ACTION SubModules_Action:
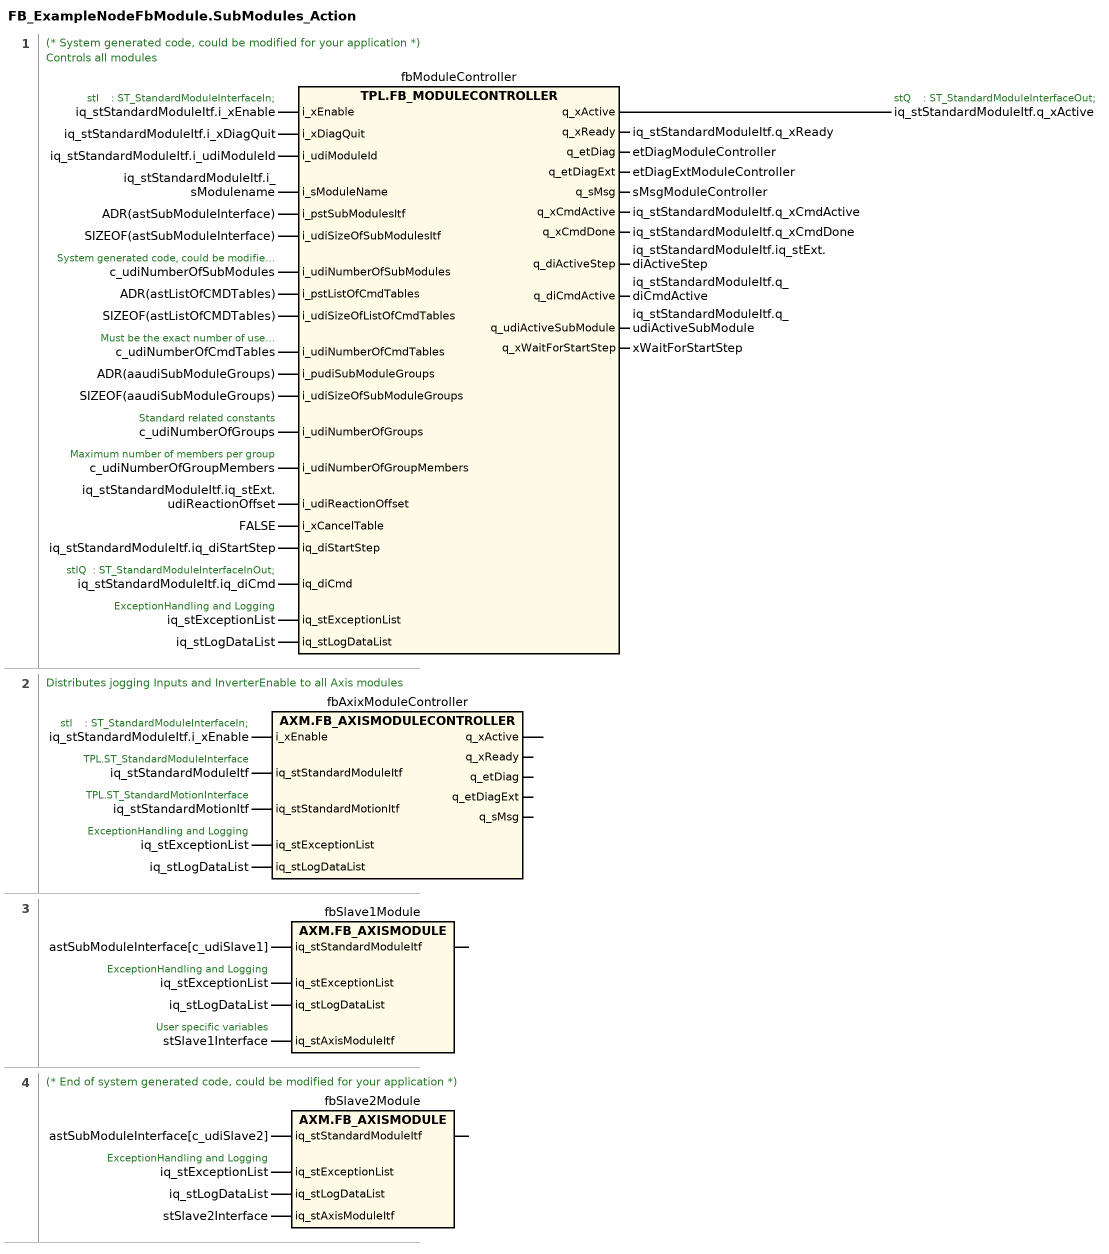
// NETWORK 1
// 					(* System generated code, could be modified for your application *)
// Controls all modules
//
//   fbModuleController: Modules related variables
//   iq_stStandardModuleItf.i_xEnable: stI : ST_StandardModuleInterfaceIn;
//   c_udiNumberOfSubModules: System generated code, could be modified for your application
//   c_udiNumberOfCmdTables: Must be the exact number of used CMDTables!
//   c_udiNumberOfGroups: Standard related constants
//   c_udiNumberOfGroupMembers: Maximum number of members per group
//   iq_stStandardModuleItf.iq_diCmd: stIQ : ST_StandardModuleInterfaceInOut;
//   iq_stExceptionList: ExceptionHandling and Logging
//   iq_stStandardModuleItf.q_xActive: stQ : ST_StandardModuleInterfaceOut;
fbModuleController(
    i_xEnable := iq_stStandardModuleItf.i_xEnable,
    i_xDiagQuit := iq_stStandardModuleItf.i_xDiagQuit,
    i_udiModuleId := iq_stStandardModuleItf.i_udiModuleId,
    i_sModuleName := iq_stStandardModuleItf.i_sModulename,
    i_pstSubModulesItf := ADR(astSubModuleInterface),
    i_udiSizeOfSubModulesItf := SIZEOF(astSubModuleInterface),
    i_udiNumberOfSubModules := c_udiNumberOfSubModules,
    i_pstListOfCmdTables := ADR(astListOfCMDTables),
    i_udiSizeOfListOfCmdTables := SIZEOF(astListOfCMDTables),
    i_udiNumberOfCmdTables := c_udiNumberOfCmdTables,
    i_pudiSubModuleGroups := ADR(aaudiSubModuleGroups),
    i_udiSizeOfSubModuleGroups := SIZEOF(aaudiSubModuleGroups),
    i_udiNumberOfGroups := c_udiNumberOfGroups,
    i_udiNumberOfGroupMembers := c_udiNumberOfGroupMembers,
    i_udiReactionOffset := iq_stStandardModuleItf.iq_stExt.udiReactionOffset,
    i_xCancelTable := FALSE,
    iq_diStartStep := iq_stStandardModuleItf.iq_diStartStep,
    iq_diCmd := iq_stStandardModuleItf.iq_diCmd,
    iq_stExceptionList := iq_stExceptionList,
    iq_stLogDataList := iq_stLogDataList,
    q_xReady => iq_stStandardModuleItf.q_xReady,
    q_etDiag => etDiagModuleController,
    q_etDiagExt => etDiagExtModuleController,
    q_sMsg => sMsgModuleController,
    q_xCmdActive => iq_stStandardModuleItf.q_xCmdActive,
    q_xCmdDone => iq_stStandardModuleItf.q_xCmdDone,
    q_diActiveStep => iq_stStandardModuleItf.iq_stExt.diActiveStep,
    q_diCmdActive => iq_stStandardModuleItf.q_diCmdActive,
    q_udiActiveSubModule => iq_stStandardModuleItf.q_udiActiveSubModule,
    q_xWaitForStartStep => xWaitForStartStep); // TPL.FB_MODULECONTROLLER
iq_stStandardModuleItf.q_xActive := fbModuleController.q_xActive;

// NETWORK 2
// Distributes jogging Inputs and InverterEnable to all Axis modules
//   iq_stStandardModuleItf.i_xEnable: stI : ST_StandardModuleInterfaceIn;
//   iq_stStandardModuleItf: TPL.ST_StandardModuleInterface
//   iq_stStandardMotionItf: TPL.ST_StandardMotionInterface
//   iq_stExceptionList: ExceptionHandling and Logging
fbAxixModuleController(
    i_xEnable := iq_stStandardModuleItf.i_xEnable,
    iq_stStandardModuleItf := iq_stStandardModuleItf,
    iq_stStandardMotionItf := iq_stStandardMotionItf,
    iq_stExceptionList := iq_stExceptionList,
    iq_stLogDataList := iq_stLogDataList); // AXM.FB_AXISMODULECONTROLLER

// NETWORK 3
//   iq_stExceptionList: ExceptionHandling and Logging
//   stSlave1Interface: User specific variables
fbSlave1Module(
    iq_stStandardModuleItf := astSubModuleInterface[c_udiSlave1],
    iq_stExceptionList := iq_stExceptionList,
    iq_stLogDataList := iq_stLogDataList,
    iq_stAxisModuleItf := stSlave1Interface); // AXM.FB_AXISMODULE

// NETWORK 4
// (* End of system generated code, could be modified for your application *)
//   iq_stExceptionList: ExceptionHandling and Logging
fbSlave2Module(
    iq_stStandardModuleItf := astSubModuleInterface[c_udiSlave2],
    iq_stExceptionList := iq_stExceptionList,
    iq_stLogDataList := iq_stLogDataList,
    iq_stAxisModuleItf := stSlave2Interface); // AXM.FB_AXISMODULE
END_ACTION

ACTION UpdateStructs:
(* System generated code, do not change without consulting 'Schneider Electric Automation GmbH' - otherwise you risk instability!!!*)
fbDetectOnlineChange(	i_xEnable	:= TRUE, 
						i_xDetect	:= TRUE, 
						q_xActive	=> xDetectOnlineChangeActive, 
						q_xReady	=> xDetectOnlineChangeReady, 
						q_etDiag	=> etDetectOnlineChangeDiag, 
						q_etDiagExt	=> etDetectOnlineChangeDiagExt, 
						q_sMsg		=> sDetectOnlineChangeMsg, 
						q_xChange	=> );
						
IF(NOT fbDetectOnlineChange.q_xChange) THEN
	RETURN;
END_IF

iq_stStandardModuleItf.iq_stExt.udiNumberOfSubModules 	:= c_udiNumberOfSubModules;
iq_stStandardModuleItf.iq_stExt.dwSubModulesItf		 	:= ADR(astSubModuleInterface);
iq_stStandardModuleItf.iq_stExt.pdwSubModulesAddItf 	:= ADR(adwSubModuleAddInterfaces);
iq_stStandardModuleItf.iq_stExt.pstListOfCmdTables		:= ADR(astListOfCmdTables);
iq_stStandardModuleItf.iq_stExt.udiNumberOfCmdTables	:= c_udiNumberOfCmdTables;
(* End of system generated code, do not change without consulting 'Schneider Electric Automation GmbH' - otherwise you risk instability!!!*)

(* System generated code, could be modified for your application *)
xUpdateStructsException := FALSE;

(*****************************************************************************************************************************************************)
(* Update CmdTable - Prepare *)

TPL.FC_UpdateCmdTableListElement(	i_pstListofCmdTables	:= ADR(astListOfCmdTables),
									i_udiNumberOfCmdTables	:= c_udiNumberOfCmdTables,
									i_diCmd					:= ET_Cmd.Prepare,
									i_pstCmdTable			:= ADR(astPrepareTable),
									q_etDiag				=> etDiag,
									q_etDiagExt				=> etDiagExtTPL);
									
IF etDiag <> GD.ET_Diag.Ok AND NOT xUpdateStructsException THEN
	xUpdateStructsException := TRUE;
	
	stUpdateStructsException.sMsg := PDL.FC_MultiConcat(i_sString1 := 'Update CmdTable: Prepare - ', 
														i_sString2 := GD.FC_EtDiagToString(i_etDiag := etDiag), 
														i_sString3 := ' - ', 
														i_sString4 := TPL.FC_EtDiagExtToString(i_etDiagExt := etDiagExtTPL));
END_IF										

(*****************************************************************************************************************************************************)
(* Update CmdTable - Auto *)

TPL.FC_UpdateCmdTableListElement(	i_pstListofCmdTables	:= ADR(astListOfCmdTables),
									i_udiNumberOfCmdTables	:= c_udiNumberOfCmdTables,
									i_diCmd					:= ET_Cmd.Auto,
									i_pstCmdTable			:= ADR(astAutoTable),
									q_etDiag				=> etDiag,
									q_etDiagExt				=> etDiagExtTPL);
									
IF etDiag <> GD.ET_Diag.Ok AND NOT xUpdateStructsException THEN
	xUpdateStructsException := TRUE;
	
	stUpdateStructsException.sMsg := PDL.FC_MultiConcat(i_sString1 := 'Update CmdTable: Auto - ', 
														i_sString2 := GD.FC_EtDiagToString(i_etDiag := etDiag), 
														i_sString3 := ' - ', 
														i_sString4 := TPL.FC_EtDiagExtToString(i_etDiagExt := etDiagExtTPL));
END_IF		

(*****************************************************************************************************************************************************)
(* Update CmdTable - Manual *)

TPL.FC_UpdateCmdTableListElement(	i_pstListofCmdTables	:= ADR(astListOfCmdTables),
									i_udiNumberOfCmdTables	:= c_udiNumberOfCmdTables,
									i_diCmd					:= ET_Cmd.Manual,
									i_pstCmdTable			:= ADR(astManualTable),
									q_etDiag				=> etDiag,
									q_etDiagExt				=> etDiagExtTPL);
									
IF etDiag <> GD.ET_Diag.Ok AND NOT xUpdateStructsException THEN
	xUpdateStructsException := TRUE;
	
	stUpdateStructsException.sMsg := PDL.FC_MultiConcat(i_sString1 := 'Update CmdTable: Manual - ', 
														i_sString2 := GD.FC_EtDiagToString(i_etDiag := etDiag), 
														i_sString3 := ' - ', 
														i_sString4 := TPL.FC_EtDiagExtToString(i_etDiagExt := etDiagExtTPL));
END_IF		

(*****************************************************************************************************************************************************)
(* Update CmdTable - Stop *)

TPL.FC_UpdateCmdTableListElement(	i_pstListofCmdTables	:= ADR(astListOfCmdTables),
									i_udiNumberOfCmdTables	:= c_udiNumberOfCmdTables,
									i_diCmd					:= ET_Cmd.Stop,
									i_pstCmdTable			:= ADR(astStopTable),
									q_etDiag				=> etDiag,
									q_etDiagExt				=> etDiagExtTPL);
									
IF etDiag <> GD.ET_Diag.Ok AND NOT xUpdateStructsException THEN
	xUpdateStructsException := TRUE;
	
	stUpdateStructsException.sMsg := PDL.FC_MultiConcat(i_sString1 := 'Update CmdTable: Stop - ', 
														i_sString2 := GD.FC_EtDiagToString(i_etDiag := etDiag), 
														i_sString3 := ' - ', 
														i_sString4 := TPL.FC_EtDiagExtToString(i_etDiagExt := etDiagExtTPL));
END_IF		

(*****************************************************************************************************************************************************)
(* Update CmdTable - Start *)

TPL.FC_UpdateCmdTableListElement(	i_pstListofCmdTables	:= ADR(astListOfCmdTables),
									i_udiNumberOfCmdTables	:= c_udiNumberOfCmdTables,
									i_diCmd					:= ET_Cmd.Start,
									i_pstCmdTable			:= ADR(astStartTable),
									q_etDiag				=> etDiag,
									q_etDiagExt				=> etDiagExtTPL);
									
IF etDiag <> GD.ET_Diag.Ok AND NOT xUpdateStructsException THEN
	xUpdateStructsException := TRUE;
	
	stUpdateStructsException.sMsg := PDL.FC_MultiConcat(i_sString1 := 'Update CmdTable: Start - ', 
														i_sString2 := GD.FC_EtDiagToString(i_etDiag := etDiag), 
														i_sString3 := ' - ', 
														i_sString4 := TPL.FC_EtDiagExtToString(i_etDiagExt := etDiagExtTPL));
END_IF		

(*****************************************************************************************************************************************************)
(* Update CmdTable - Abort *)

TPL.FC_UpdateCmdTableListElement(	i_pstListofCmdTables	:= ADR(astListOfCmdTables),
									i_udiNumberOfCmdTables	:= c_udiNumberOfCmdTables,
									i_diCmd					:= ET_Cmd.Abort,
									i_pstCmdTable			:= ADR(astAbortTable),
									q_etDiag				=> etDiag,
									q_etDiagExt				=> etDiagExtTPL);
									
IF etDiag <> GD.ET_Diag.Ok AND NOT xUpdateStructsException THEN
	xUpdateStructsException := TRUE;
	
	stUpdateStructsException.sMsg := PDL.FC_MultiConcat(i_sString1 := 'Update CmdTable: Abort - ', 
														i_sString2 := GD.FC_EtDiagToString(i_etDiag := etDiag), 
														i_sString3 := ' - ', 
														i_sString4 := TPL.FC_EtDiagExtToString(i_etDiagExt := etDiagExtTPL));
END_IF		

(*****************************************************************************************************************************************************)
(* Update CmdTable - Hold *)

TPL.FC_UpdateCmdTableListElement(	i_pstListofCmdTables	:= ADR(astListOfCmdTables),
									i_udiNumberOfCmdTables	:= c_udiNumberOfCmdTables,
									i_diCmd					:= ET_Cmd.Hold,
									i_pstCmdTable			:= ADR(astHoldTable),
									q_etDiag				=> etDiag,
									q_etDiagExt				=> etDiagExtTPL);
									
IF etDiag <> GD.ET_Diag.Ok AND NOT xUpdateStructsException THEN
	xUpdateStructsException := TRUE;
	
	stUpdateStructsException.sMsg := PDL.FC_MultiConcat(i_sString1 := 'Update CmdTable: Hold - ', 
														i_sString2 := GD.FC_EtDiagToString(i_etDiag := etDiag), 
														i_sString3 := ' - ', 
														i_sString4 := TPL.FC_EtDiagExtToString(i_etDiagExt := etDiagExtTPL));
END_IF		

(*****************************************************************************************************************************************************)
(* Update CmdTable - BrakeRelease *)

TPL.FC_UpdateCmdTableListElement(	i_pstListofCmdTables	:= ADR(astListOfCmdTables),
									i_udiNumberOfCmdTables	:= c_udiNumberOfCmdTables,
									i_diCmd					:= ET_Cmd.BrakeRelease,
									i_pstCmdTable			:= ADR(astBrakeReleaseTable),
									q_etDiag				=> etDiag,
									q_etDiagExt				=> etDiagExtTPL);
									
IF etDiag <> GD.ET_Diag.Ok AND NOT xUpdateStructsException THEN
	xUpdateStructsException := TRUE;
	
	stUpdateStructsException.sMsg := PDL.FC_MultiConcat(i_sString1 := 'Update CmdTable: BrakeRelease - ', 
														i_sString2 := GD.FC_EtDiagToString(i_etDiag := etDiag), 
														i_sString3 := ' - ', 
														i_sString4 := TPL.FC_EtDiagExtToString(i_etDiagExt := etDiagExtTPL));
END_IF		
									
(*****************************************************************************************************************************************************)
(* Update AddInterface - Slave1 *)

AXM.FC_UpdateAddInterfaceStruct(	i_pdwSubModuleAddInterfaces	:= ADR(adwSubModuleAddInterfaces),
									i_udiSubModuleConstant		:= c_udiSlave1,
									iq_stAxisModuleItf			:= stSlave1Interface,
									q_etDiag					=> etDiag,
									q_etDiagExt					=> etDiagExtAXM);
									
IF etDiag <> GD.ET_Diag.Ok AND NOT xUpdateStructsException THEN
	xUpdateStructsException := TRUE;
	
	stUpdateStructsException.sMsg := PDL.FC_MultiConcat(i_sString1 := 'Update AddInterface: Slave1 - ', 
														i_sString2 := GD.FC_EtDiagToString(i_etDiag := etDiag), 
														i_sString3 := ' - ', 
														i_sString4 := AXM.FC_EtDiagExtToString(i_etDiagExt := etDiagExtAXM));
END_IF		

(*****************************************************************************************************************************************************)
(* Update AddInterface - Slave2 *)

AXM.FC_UpdateAddInterfaceStruct(	i_pdwSubModuleAddInterfaces	:= ADR(adwSubModuleAddInterfaces),
									i_udiSubModuleConstant		:= c_udiSlave2,
									iq_stAxisModuleItf			:= stSlave2Interface,
									q_etDiag					=> etDiag,
									q_etDiagExt					=> etDiagExtAXM);
									
IF etDiag <> GD.ET_Diag.Ok AND NOT xUpdateStructsException THEN
	xUpdateStructsException := TRUE;
	
	stUpdateStructsException.sMsg := PDL.FC_MultiConcat(i_sString1 := 'Update AddInterface: Slave2 - ', 
														i_sString2 := GD.FC_EtDiagToString(i_etDiag := etDiag), 
														i_sString3 := ' - ', 
														i_sString4 := AXM.FC_EtDiagExtToString(i_etDiagExt := etDiagExtAXM));
END_IF		

(*****************************************************************************************************************************************************)
(* Set exception if any exception occurred *)

TPL.FC_SetException(i_xExceptionActive	:= xUpdateStructsException, 
					iq_stException		:= stUpdateStructsException, 
					iq_stExceptionList	:= iq_stExceptionList, 
					iq_stLogDataList	:= iq_stLogDataList);
					
xInitSuccessful := xInitSuccessful AND NOT xUpdateStructsException;

etDiag := GD.ET_Diag.Ok;
(* End of system generated code, could be modified for your application *)
END_ACTION

END_FUNCTION_BLOCK

// LMC_PacDrive/Application/CrankModuleExample/Visualization/VIS_Main
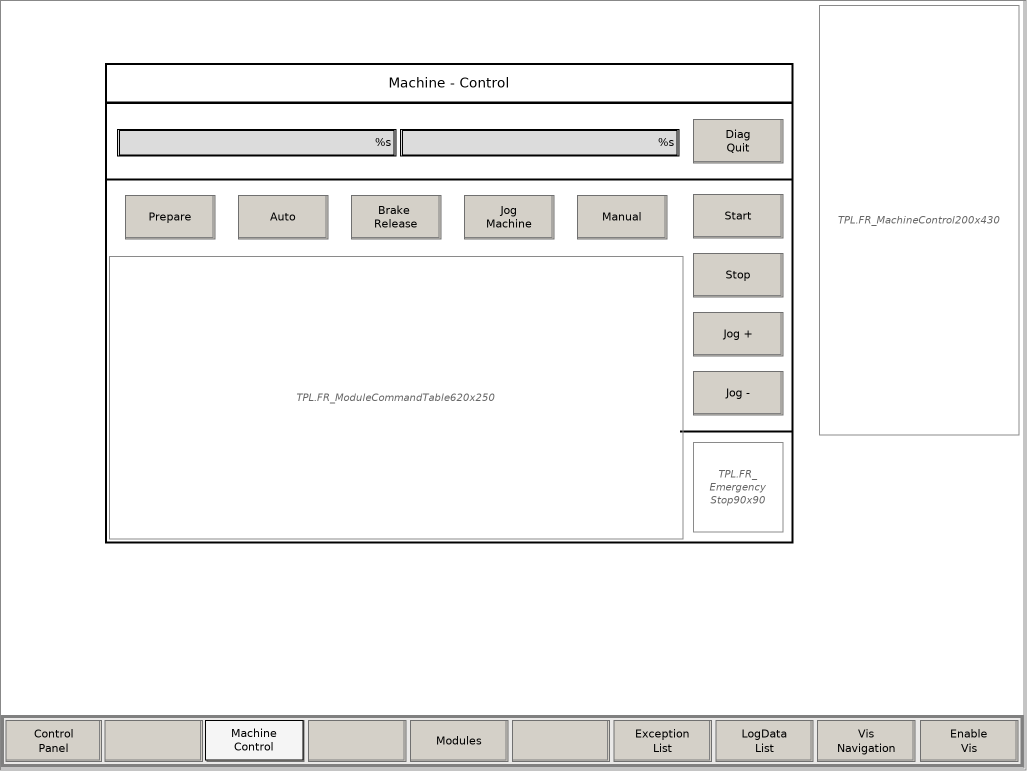
VISUALIZATION VIS_Main  // 1027x771
    Frame (0,0 1024x768)
        shows TPL.FR_NavControl1024x768(i_sTitle := 'Template')
    Rectangle (105,63 688x480)
    Rectangle (105,63 688x40), "Machine - Control"
    Rectangle (105,102 688x78)
    Textfield (400,129 279x27)
    Button (693,119 90x44), "Diag Quit", colour toggle: SR_VisControl.vpq_xMachineInException
        p573394764: SR_VisControl.vpq_dwDiagQuitColor
        tap G_xDiagQuitEpas
    Textfield (117,129 279x27)
    Rectangle (402,130 275x25), "%s", text variable: SR_VisControl.vpq_etMainModuleControllerDiagExt, colour toggle: SR_VisControl.vpq_xMachineInException
        p2167032090: SR_VisControl.vpq_dwDiagQuitColor
    Rectangle (119,130 275x25), "%s", text variable: SR_VisControl.vpq_etMainModuleControllerDiag, colour toggle: SR_VisControl.vpq_xMachineInException
        p2167032090: SR_VisControl.vpq_dwDiagQuitColor
    Button (693,194 90x44), "Start", colour toggle: G_xStartEpas
        tap G_xStartEpas
    Button (693,253 90x44), "Stop", colour toggle: G_xStopEpas
        tap G_xStopEpas p3779583253=TRUE
    Button (693,312 90x44), "Jog +", colour toggle: G_xJogForwEpas
        tap G_xJogForwEpas p3779583253=TRUE
    Button (693,371 90x44), "Jog -", colour toggle: G_xJogBackEpas
        tap G_xJogBackEpas p3779583253=TRUE
    Button (125,195 90x44), "Prepare", colour toggle: G_xPrepareActive
        tap G_xDoPrepare
    Button (238,195 90x44), "Auto", colour toggle: G_xAutoActive
        tap G_xDoAuto
    Button (351,195 90x44), "Brake Release", colour toggle: G_xBrakeReleaseActive
        tap G_xDoBrakeRelease
    Button (464,195 90x44), "Jog Machine", colour toggle: G_xJogMachineActive
        tap G_xDoJogMachine
    Button (577,195 90x44), "Manual", colour toggle: G_xManualActive
        tap G_xDoManual
    Polyline (680,431) (793,431)
    Frame (693,442 90x90)
        shows TPL.FR_EmergencyStop90x90(i_xChangeColor := NOT G_xEmergencyEpas, i_xInvisible := FALSE, iq_xToggle := G_xEmergencyEpas)
    Frame (109,256 574x283)
        shows TPL.FR_ModuleCommandTable620x250(i_stCurrentModuleStandardItf := SR_VisControl.vpq_stMachineInterface, i_astActualCmdTable := SR_VisControl.vpq_astActualCmdTableMain, i_udiNumberOfCmdSteps := SR_VisControl.vpq_udiNumberOfCmdStepsMain, i_sCmdTitel := SR_VisControl.vpq_sCmdTitelMain, i_xDoEnable := SR_VisControl.vpq_xDoEnable, i_xDisableScrollUp := SR_VisControl.vpq_xDisableScrollUpMain, i_xDisableScrollDown := SR_VisControl.vpq_xDisableScrollDownMain, iq_udiIndexMin := SR_VisControl.vpiq_udiIndexMinMain)
        p2190627833: SR_VisControl.vpq_stMachineInterface
        p3492251336: SR_VisControl.vpq_stMachineInterface.iq_stExt.diActiveStep
    Frame (1,715 1024x54)
        shows FR_NavigationButtons()
    Rectangle (205,720 98x40), "Machine Control"
    Frame (819,5 200x430), invisible if: NOT SR_VisControl.vpiq_xShowControlFrame
        shows TPL.FR_MachineControl200x430(i_stMachineItf := SR_VisControl.vpq_stMachineInterface, i_xPrepareActive := G_xPrepareActive, i_xAutoActive := G_xAutoActive, i_xBrakeReleaseActive := G_xBrakeReleaseActive, i_xJogMachineActive := G_xJogMachineActive, i_xManualActive := G_xManualActive, i_xException := SR_VisControl.vpq_xMachineInException, i_dwDiagQuitColor := SR_VisControl.vpq_dwDiagQuitColor, iq_iPositionX := SR_VisControl.vpiq_iPositionX, iq_iPositionY := SR_VisControl.vpiq_iPositionY, iq_xEmergencyEpas := G_xEmergencyEpas, iq_xStartEpas := G_xStartEpas, iq_xStopEpas := G_xStopEpas, iq_xJogForwEpas := G_xJogForwEpas, iq_xJogBackEpas := G_xJogBackEpas, iq_xDoPrepare := G_xDoPrepare, iq_xDoAuto := G_xDoAuto, iq_xDoBrakeRelease := G_xDoBrakeRelease, iq_xDoJogMachine := G_xDoJogMachine, iq_xDoManual := G_xDoManual, iq_xDiagQuitEpas := G_xDiagQuitEpas)
        p1457045297: SR_VisControl.stMachineInterface.stQ.xError
        p1941967854: g_I_xEmergency_Epas
        p2531571229: g_I_xStart_Epas
        p1511842254: g_I_xStop_Epas
        p745511063: g_I_xJogForw_Epas
        p3518271027: g_I_xJogBack_Epas
        p1982879521: g_I_xErrorQuit_Epas
        p3866886353: SR_VisControl.dwErrorQuitColor
        p1761348311: SR_VisControl.vpq_stMachineInterface
        p3560616238: SR_VisControl.vpiq_iPositionX
        p2738717112: SR_VisControl.vpiq_iPositionY
END_VISUALIZATION

// LMC_PacDrive/Application/CrankModuleExample/Visualization/CrankModule/VIS_CrankModule
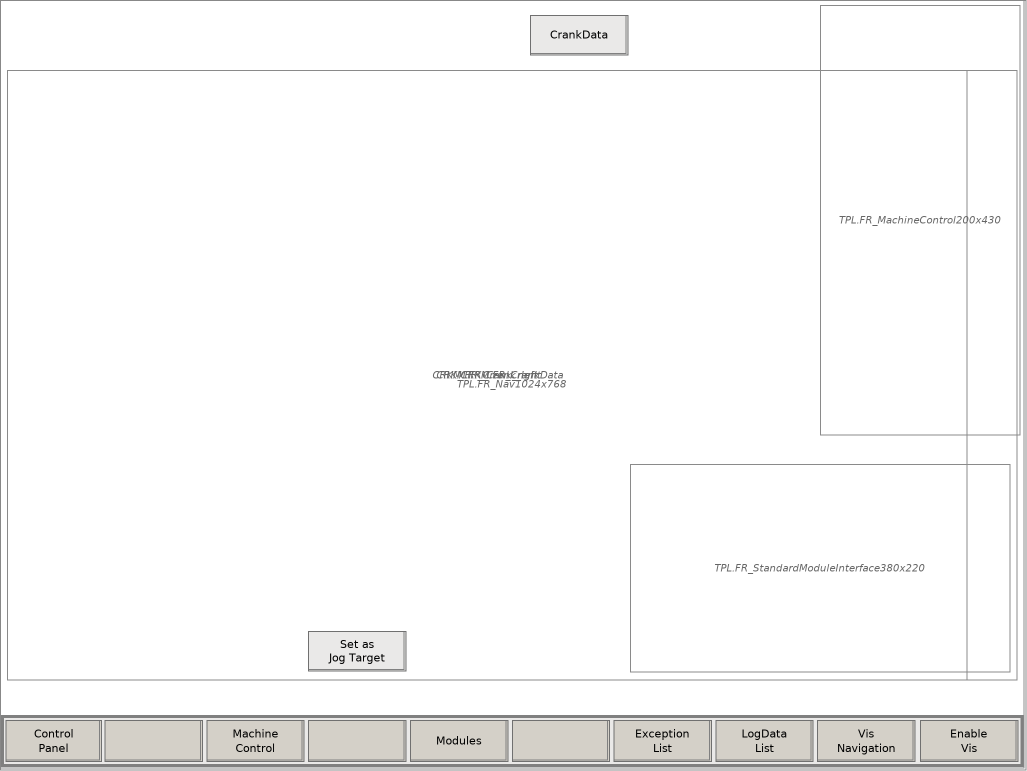
VISUALIZATION VIS_CrankModule  // 1027x771
    Frame (0,0 1024x768)
        shows TPL.FR_Nav1024x768(i_sTitle := 'CrankModule')
    Frame (7,70 960x610), invisible if: NOT SR_VisControl.vpq_xFrameSetCrankLeftInvisible
        shows CRKM.FR_Crank_right(iq_fbCrankModuleVisController := SR_VisControl.vpiq_fbCrankModuleVisController)
    Frame (7,70 960x610), invisible if: SR_VisControl.vpq_xFrameSetCrankLeftInvisible
        shows CRKM.FR_Crank_left(iq_fbCrankModuleVisController := SR_VisControl.vpiq_fbCrankModuleVisController)
    Frame (7,70 1010x610), invisible if: SR_VisControl.vpq_xFrameCrankDataInvisible
        shows CRKM.FR_CrankData(iq_fbCrankModuleVisController := SR_VisControl.vpiq_fbCrankModuleVisController)
    Frame (630,464 380x208), invisible if: SR_VisControl.vpq_xFrameCrankDataInvisible
        shows TPL.FR_StandardModuleInterface380x220(i_stCurrentModuleStandardItf := SR_VisControl.vpq_stCurrentModuleStandardInterface, i_sCurrentModuleReaction := SR_VisControl.vpq_sCurrentModuleReaction, i_udiModuleReactionIndexMin := SR_VisControl.vpq_udiModuleReactionIndexMin, i_axModuleReaction := SR_VisControl.vpq_axModuleReaction, i_udiNumberOfReactions := TPL.Gc_udiMaxNumberOfReactions, iq_xModuleReactionDown := SR_VisControl.vpiq_xModuleReactionDown, iq_xModuleReactionUp := SR_VisControl.vpiq_xModuleReactionUp, iq_diStartStepToSet := SR_VisControl.vpiq_diStartStepToSet, iq_diCmdToSet := SR_VisControl.vpiq_diCmdToSet, iq_xEnableModuleClicked := SR_VisControl.vpiq_xEnableModuleClicked, iq_xSetCmdClicked := SR_VisControl.vpiq_xSetCmdClicked, iq_fbVisContExHandling := SR_VisControl.vpiq_fbVisContExHandling)
        p1094400588: SR_VisControl.IFB_AxisModuleVisController.xCurrentIsOfMyType
        p3339340907: ''
        p1029787830: SR_VisControl.fbVisContExHandling
        p2258115317: SR_VisControl.iModuleErrorReactionIndexMin
        p2777435286: SR_VisControl.axModuleErrorReaction
        p214250784: TPC_Gc_diMaxNumberOfErrorReactions
        p311732222: SR_VisControl.stCurrentModuleStandardInterface
        p640132070: SR_VisControl.xModuleErrorReactionDown
        p4234372197: SR_VisControl.xModuleErrorReactionUp
        p2938682392: SR_VisControl.xEnableModule_Clicked
        p3592490199: SR_VisControl.xSetCmd_Clicked
        p2307280719: SR_VisControl.stCurrentModuleStandardInterface
        p2190627833: SR_VisControl.vpq_stCurrentModuleStandardInterface
    Frame (1,715 1024x54)
        shows FR_NavigationButtons()
    Button (530,15 98x40), "CrankData", colour toggle: SR_VisControl.vpq_xFrameCrankDataInvisible
        toggle SR_VisControl.vpq_xFrameCrankDataInvisible
    Button (308,631 98x40), "Set as Jog Target", colour toggle: SR_VisControl.vpq_xCurrentIsJogTarget, invisible if: SR_VisControl.vpq_xButtonSetJogTargetInvisible
        tap SR_VisControl.vpiq_xButtonSetCurrentAsJogTarget
    Frame (820,5 200x430), invisible if: NOT SR_VisControl.vpiq_xShowControlFrame
        shows TPL.FR_MachineControl200x430(i_stMachineItf := SR_VisControl.vpq_stMachineInterface, i_xPrepareActive := G_xPrepareActive, i_xAutoActive := G_xAutoActive, i_xBrakeReleaseActive := G_xBrakeReleaseActive, i_xJogMachineActive := G_xJogMachineActive, i_xManualActive := G_xManualActive, i_xException := SR_VisControl.vpq_xMachineInException, i_dwDiagQuitColor := SR_VisControl.vpq_dwDiagQuitColor, iq_iPositionX := SR_VisControl.vpiq_iPositionX, iq_iPositionY := SR_VisControl.vpiq_iPositionY, iq_xEmergencyEpas := G_xEmergencyEpas, iq_xStartEpas := G_xStartEpas, iq_xStopEpas := G_xStopEpas, iq_xJogForwEpas := G_xJogForwEpas, iq_xJogBackEpas := G_xJogBackEpas, iq_xDoPrepare := G_xDoPrepare, iq_xDoAuto := G_xDoAuto, iq_xDoBrakeRelease := G_xDoBrakeRelease, iq_xDoJogMachine := G_xDoJogMachine, iq_xDoManual := G_xDoManual, iq_xDiagQuitEpas := G_xDiagQuitEpas)
        p1457045297: SR_VisControl.stMachineInterface.stQ.xError
        p1941967854: g_I_xEmergency_Epas
        p2531571229: g_I_xStart_Epas
        p1511842254: g_I_xStop_Epas
        p745511063: g_I_xJogForw_Epas
        p3518271027: g_I_xJogBack_Epas
        p1982879521: g_I_xErrorQuit_Epas
        p3866886353: SR_VisControl.dwErrorQuitColor
        p1761348311: SR_VisControl.vpq_stMachineInterface
        p3560616238: SR_VisControl.vpiq_iPositionX
        p2738717112: SR_VisControl.vpiq_iPositionY
END_VISUALIZATION

// LMC_PacDrive/Application/FR_ButtonAssignId
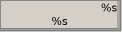
VISUALIZATION FR_ButtonAssignId  // 122x32
VAR_INPUT
	i_udiId : UDINT;
	i_sName : STRING[80];
	i_udiCurrentModuleId : UDINT;
END_VAR
VAR_IN_OUT
	iq_udiAssignTarget : UDINT;
END_VAR
    Button (0,0 120x30), "%s", text variable: i_sName, colour toggle: i_udiId = i_udiCurrentModuleId, invisible if: i_udiId<1
    Rectangle (0,0 119x29), "%s", text variable: i_udiId, invisible if: i_udiId<1
        OnMouseUp: execute { iq_udiAssignTarget := i_udiId; }
END_VISUALIZATION

// LMC_PacDrive/Application/FR_ExampleLeafModule
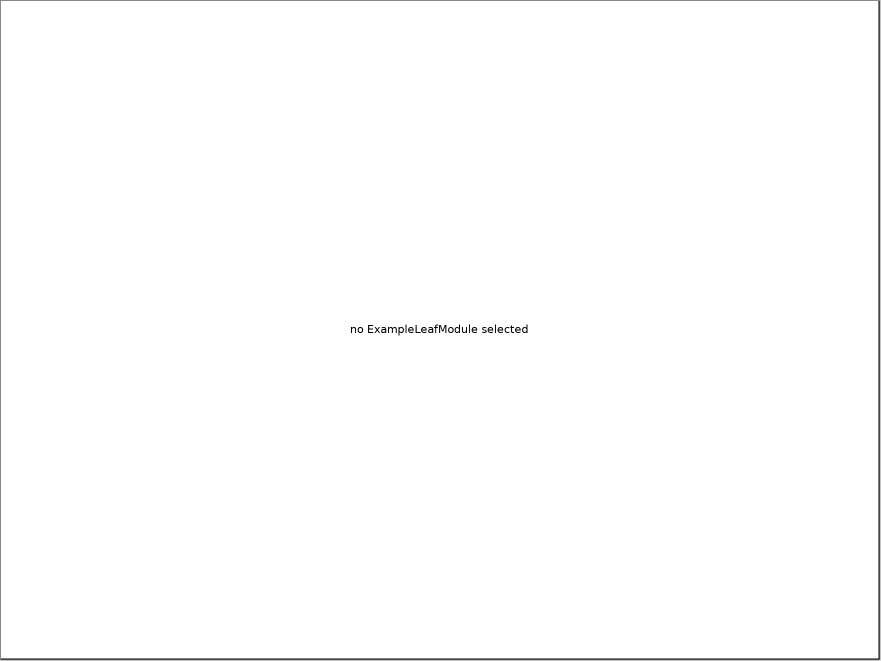
VISUALIZATION FR_ExampleLeafModule  // 881x661
VAR_IN_OUT
	iq_xModuleReactionDown				: BOOL;
	iq_xModuleReactionUp				: BOOL;
	iq_diStartStepToSet					: DINT;
	iq_diCmdToSet						: DINT;
	iq_xEnableModuleClicked				: BOOL;
	iq_xSetCmdClicked					: BOOL;
	iq_fbVisContExHandling				: TPL.FB_VisControllerExceptionHandling;
	iq_fbExampleLeafModuleVisController : FB_ExampleLeafModuleVisController;
END_VAR
VAR_INPUT
	i_stCurrentModuleStandardInterface : TPL.ST_StandardModuleInterface;
	i_sCurrentModuleReaction	: STRING[80];
	i_udiModuleReactionIndexMin : UDINT;
	i_axModuleReaction			: ARRAY [1..10] OF BOOL;
	i_udiNumberOfReactions 		: UDINT;
END_VAR
    Frame (0,0 380x211)
        shows TPL.FR_StandardModuleInterface380x220(i_stCurrentModuleStandardItf := i_stCurrentModuleStandardInterface, i_sCurrentModuleReaction := i_sCurrentModuleReaction, i_udiModuleReactionIndexMin := i_udiModuleReactionIndexMin, i_axModuleReaction := i_axModuleReaction, i_udiNumberOfReactions := i_udiNumberOfReactions, iq_xModuleReactionDown := iq_xModuleReactionDown, iq_xModuleReactionUp := iq_xModuleReactionUp, iq_diStartStepToSet := iq_diStartStepToSet, iq_diCmdToSet := iq_diCmdToSet, iq_xEnableModuleClicked := iq_xEnableModuleClicked, iq_xSetCmdClicked := iq_xSetCmdClicked, iq_fbVisContExHandling := iq_fbVisContExHandling)
        p3339340907: i_sZoomToVisModuleErrors
        p1094400588: i_xCurrentIsOfMyType
        p1029787830: i_fbVisContExHandling
        p2258115317: i_iModuleErrorReactionIndexMin
        p2777435286: i_axModuleErrorReaction
        p214250784: i_diNumberOfErrorreactions
        p311732222: iq_stCurrentModuleStandardInterface
        p640132070: iq_xModuleErrorReactionDown
        p4234372197: iq_xModuleErrorReactionUp
        p2938682392: iq_xEnableModule_Clicked
        p3592490199: iq_xSetCmd_Clicked
        p2307280719: iq_stCurrentModuleStandardInterface
        p2190627833: i_stCurrentModuleStandardInterface
    Rectangle (0,0 879x659), "no ExampleLeafModule selected", invisible if: iq_fbExampleLeafModuleVisController.xCurrentIsOfMyType
END_VISUALIZATION

// LMC_PacDrive/Application/FR_ExampleLeafModuleSelect
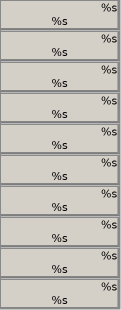
VISUALIZATION FR_ExampleLeafModuleSelect  // 121x310
VAR_IN_OUT
	iq_fbExampleLeafModuleVisController : FB_ExampleLeafModuleVisController;
END_VAR
VAR_INPUT
	i_stCurrentModuleStandardInterface : TPL.ST_StandardModuleInterface;
END_VAR
    Frame (0,0 119x29)
        shows FR_ButtonAssignId(i_udiId := iq_fbExampleLeafModuleVisController.audiExampleLeafModuleId[1], i_sName := iq_fbExampleLeafModuleVisController.asExampleLeafModuleName[1], i_udiCurrentModuleId := i_stCurrentModuleStandardInterface.i_udiModuleId, iq_udiAssignTarget := iq_fbExampleLeafModuleVisController.udiSetAsCurrentModule)
    Frame (0,31 119x29)
        shows FR_ButtonAssignId(i_udiId := iq_fbExampleLeafModuleVisController.audiExampleLeafModuleId[2], i_sName := iq_fbExampleLeafModuleVisController.asExampleLeafModuleName[2], i_udiCurrentModuleId := i_stCurrentModuleStandardInterface.i_udiModuleId, iq_udiAssignTarget := iq_fbExampleLeafModuleVisController.udiSetAsCurrentModule)
    Frame (0,62 119x29)
        shows FR_ButtonAssignId(i_udiId := iq_fbExampleLeafModuleVisController.audiExampleLeafModuleId[3], i_sName := iq_fbExampleLeafModuleVisController.asExampleLeafModuleName[3], i_udiCurrentModuleId := i_stCurrentModuleStandardInterface.i_udiModuleId, iq_udiAssignTarget := iq_fbExampleLeafModuleVisController.udiSetAsCurrentModule)
    Frame (0,93 119x29)
        shows FR_ButtonAssignId(i_udiId := iq_fbExampleLeafModuleVisController.audiExampleLeafModuleId[4], i_sName := iq_fbExampleLeafModuleVisController.asExampleLeafModuleName[4], i_udiCurrentModuleId := i_stCurrentModuleStandardInterface.i_udiModuleId, iq_udiAssignTarget := iq_fbExampleLeafModuleVisController.udiSetAsCurrentModule)
    Frame (0,124 119x29)
        shows FR_ButtonAssignId(i_udiId := iq_fbExampleLeafModuleVisController.audiExampleLeafModuleId[5], i_sName := iq_fbExampleLeafModuleVisController.asExampleLeafModuleName[5], i_udiCurrentModuleId := i_stCurrentModuleStandardInterface.i_udiModuleId, iq_udiAssignTarget := iq_fbExampleLeafModuleVisController.udiSetAsCurrentModule)
    Frame (0,155 119x29)
        shows FR_ButtonAssignId(i_udiId := iq_fbExampleLeafModuleVisController.audiExampleLeafModuleId[6], i_sName := iq_fbExampleLeafModuleVisController.asExampleLeafModuleName[6], i_udiCurrentModuleId := i_stCurrentModuleStandardInterface.i_udiModuleId, iq_udiAssignTarget := iq_fbExampleLeafModuleVisController.udiSetAsCurrentModule)
    Frame (0,186 119x29)
        shows FR_ButtonAssignId(i_udiId := iq_fbExampleLeafModuleVisController.audiExampleLeafModuleId[7], i_sName := iq_fbExampleLeafModuleVisController.asExampleLeafModuleName[7], i_udiCurrentModuleId := i_stCurrentModuleStandardInterface.i_udiModuleId, iq_udiAssignTarget := iq_fbExampleLeafModuleVisController.udiSetAsCurrentModule)
    Frame (0,217 119x29)
        shows FR_ButtonAssignId(i_udiId := iq_fbExampleLeafModuleVisController.audiExampleLeafModuleId[8], i_sName := iq_fbExampleLeafModuleVisController.asExampleLeafModuleName[8], i_udiCurrentModuleId := i_stCurrentModuleStandardInterface.i_udiModuleId, iq_udiAssignTarget := iq_fbExampleLeafModuleVisController.udiSetAsCurrentModule)
    Frame (0,248 119x29)
        shows FR_ButtonAssignId(i_udiId := iq_fbExampleLeafModuleVisController.audiExampleLeafModuleId[9], i_sName := iq_fbExampleLeafModuleVisController.asExampleLeafModuleName[9], i_udiCurrentModuleId := i_stCurrentModuleStandardInterface.i_udiModuleId, iq_udiAssignTarget := iq_fbExampleLeafModuleVisController.udiSetAsCurrentModule)
    Frame (0,279 119x29)
        shows FR_ButtonAssignId(i_udiId := iq_fbExampleLeafModuleVisController.audiExampleLeafModuleId[10], i_sName := iq_fbExampleLeafModuleVisController.asExampleLeafModuleName[10], i_udiCurrentModuleId := i_stCurrentModuleStandardInterface.i_udiModuleId, iq_udiAssignTarget := iq_fbExampleLeafModuleVisController.udiSetAsCurrentModule)
END_VISUALIZATION

// LMC_PacDrive/Application/VIS_ExampleLeafModule
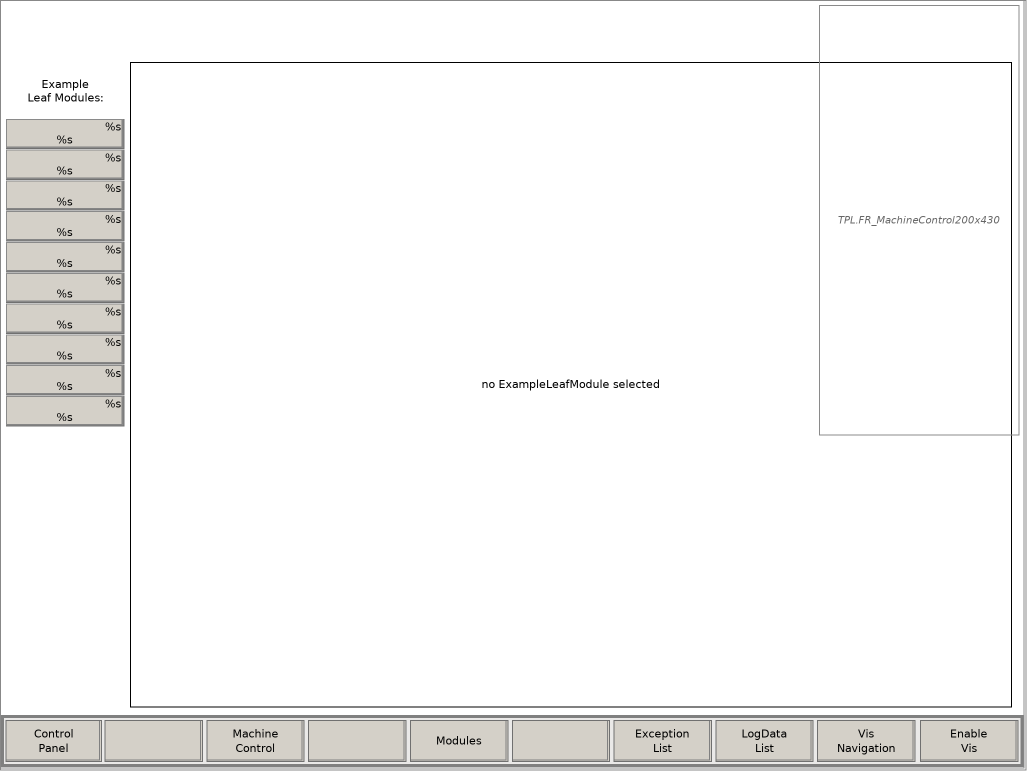
VISUALIZATION VIS_ExampleLeafModule  // 1027x771
    Frame (0,0 1024x768)
        shows TPL.FR_Nav1024x768(i_sTitle := 'Example Leaf Module')
    Frame (6,119 119x308)
        shows FR_ExampleLeafModuleSelect(i_stCurrentModuleStandardInterface := SR_VisControl.vpq_stCurrentModuleStandardInterface, iq_fbExampleLeafModuleVisController := SR_VisControl.vpiq_fbExampleLeafModuleVisController)
    Rectangle (6,65 119x52), "Example Leaf Modules:"
    Frame (130,62 884x647)
        shows FR_ExampleLeafModule(i_stCurrentModuleStandardInterface := SR_VisControl.vpq_stCurrentModuleStandardInterface, i_sCurrentModuleReaction := SR_VisControl.vpq_sCurrentModuleReaction, i_udiModuleReactionIndexMin := SR_VisControl.vpq_udiModuleReactionIndexMin, i_axModuleReaction := SR_VisControl.vpq_axModuleReaction, i_udiNumberOfReactions := TPL.Gc_udiMaxNumberOfReactions, iq_xModuleReactionDown := SR_VisControl.vpiq_xModuleReactionDown, iq_xModuleReactionUp := SR_VisControl.vpiq_xModuleReactionUp, iq_diStartStepToSet := SR_VisControl.vpiq_diStartStepToSet, iq_diCmdToSet := SR_VisControl.vpiq_diCmdToSet, iq_xEnableModuleClicked := SR_VisControl.vpiq_xEnableModuleClicked, iq_xSetCmdClicked := SR_VisControl.vpiq_xSetCmdClicked, iq_fbVisContExHandling := SR_VisControl.vpiq_fbVisContExHandling, iq_fbExampleLeafModuleVisController := SR_VisControl.vpiq_fbExampleLeafModuleVisController)
    Frame (1,715 1024x54)
        shows FR_NavigationButtons()
    Frame (819,5 200x430), invisible if: NOT SR_VisControl.vpiq_xShowControlFrame
        shows TPL.FR_MachineControl200x430(i_stMachineItf := SR_VisControl.vpq_stMachineInterface, i_xPrepareActive := G_xPrepareActive, i_xAutoActive := G_xAutoActive, i_xBrakeReleaseActive := G_xBrakeReleaseActive, i_xJogMachineActive := G_xJogMachineActive, i_xManualActive := G_xManualActive, i_xException := SR_VisControl.vpq_xMachineInException, i_dwDiagQuitColor := SR_VisControl.vpq_dwDiagQuitColor, iq_iPositionX := SR_VisControl.vpiq_iPositionX, iq_iPositionY := SR_VisControl.vpiq_iPositionY, iq_xEmergencyEpas := G_xEmergencyEpas, iq_xStartEpas := G_xStartEpas, iq_xStopEpas := G_xStopEpas, iq_xJogForwEpas := G_xJogForwEpas, iq_xJogBackEpas := G_xJogBackEpas, iq_xDoPrepare := G_xDoPrepare, iq_xDoAuto := G_xDoAuto, iq_xDoBrakeRelease := G_xDoBrakeRelease, iq_xDoJogMachine := G_xDoJogMachine, iq_xDoManual := G_xDoManual, iq_xDiagQuitEpas := G_xDiagQuitEpas)
        p1457045297: SR_VisControl.stMachineInterface.stQ.xError
        p1941967854: g_I_xEmergency_Epas
        p2531571229: g_I_xStart_Epas
        p1511842254: g_I_xStop_Epas
        p745511063: g_I_xJogForw_Epas
        p3518271027: g_I_xJogBack_Epas
        p1982879521: g_I_xErrorQuit_Epas
        p3866886353: SR_VisControl.dwErrorQuitColor
        p1761348311: SR_VisControl.vpq_stMachineInterface
        p3560616238: SR_VisControl.vpiq_iPositionX
        p2738717112: SR_VisControl.vpiq_iPositionY
END_VISUALIZATION

// LMC_PacDrive/Application/FR_ControlModuleTypes
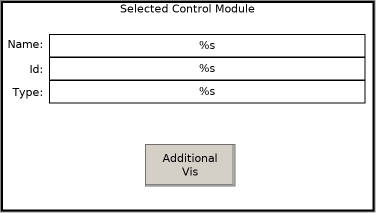
VISUALIZATION FR_ControlModuleTypes  // 376x213
VAR_INPUT
	i_sControlModuleName		: STRING[80];
	i_diControlModuleNumber		: DINT;
	i_diControlModuleType		: DINT;
END_VAR
    Rectangle (1,1 373x210), "Selected Control Module"
    Button (145,144 90x42), "Additional Vis"
        OnMouseClick:  AssignExpr=i_sZoomToControlModuleVis, Assign=VIS_ControlModule, Type=Assignment
    Textfield (49,34 316x23), "%s", text variable: i_sControlModuleName
    Rectangle (7,36 39x17), "Name:"
    Textfield (49,57 316x23), "%s", text variable: i_diControlModuleNumber
    Rectangle (7,61 39x17), "Id:"
    Rectangle (7,84 39x17), "Type:"
    Textfield (49,80 316x23), "%s", text variable: i_diControlModuleType
END_VISUALIZATION

// LMC_PacDrive/Application/FR_NavigationButtons
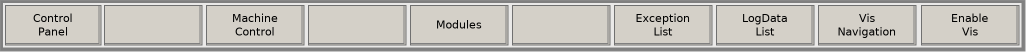
VISUALIZATION FR_NavigationButtons  // 1026x52
    Rectangle (0,0 1024x50)
    Button (410,5 98x40), "Modules"
        OnMouseClick:  Assign=VIS_Modules, Type=Assignment
    Button (5,5 96x40), "Control Panel", colour toggle: SR_VisControl.vpiq_xShowControlFrame
        toggle SR_VisControl.vpiq_xShowControlFrame
    Button (512,5 98x40)
    Button (614,5 98x40), "Exception List"
        OnMouseClick:  Assign=VIS_ExceptionList, Type=Assignment
    Button (716,5 98x40), "LogData List"
        OnMouseClick:  Assign=VIS_LogDataList, Type=Assignment
    Button (818,5 98x40), "Vis Navigation"
        OnMouseClick:  Assign=VIS_VisNavigation, Type=Assignment
    Button (308,5 98x40)
    Button (104,5 98x40)
    Button (206,5 98x40), "Machine Control"
        OnMouseClick:  Assign=VIS_Main, Type=Assignment
    Button (921,5 98x40), "Enable Vis", colour toggle: G_xDoEnableVis
        toggle G_xDoEnableVis
END_VISUALIZATION

// LMC_PacDrive/Application/FR_OtherModuleTypes
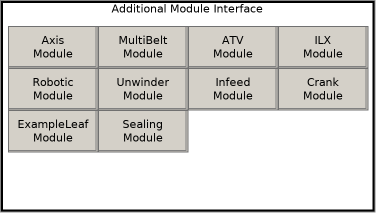
VISUALIZATION FR_OtherModuleTypes  // 376x213
    Rectangle (1,1 373x210), "Additional Module Interface"
    Button (8,26 90x42), "Axis Module", invisible if: SR_VisControl.vpq_stCurrentModuleStandardInterface.q_dwModuleType <> 3
        OnMouseClick:  Assign=VIS_AxisModule, Type=Assignment
    Button (98,26 90x42), "MultiBelt Module", invisible if: SR_VisControl.vpq_stCurrentModuleStandardInterface.q_dwModuleType <> 4
    Button (188,26 90x42), "ATV Module", invisible if: SR_VisControl.vpq_stCurrentModuleStandardInterface.q_dwModuleType <> 9
    Button (278,26 90x42), "ILX Module", invisible if: SR_VisControl.vpq_stCurrentModuleStandardInterface.q_dwModuleType <> 10
    Button (8,68 90x42), "Robotic Module", invisible if: SR_VisControl.vpq_stCurrentModuleStandardInterface.q_dwModuleType <> 6
    Button (8,110 90x42), "ExampleLeaf Module", invisible if: SR_VisControl.vpq_stCurrentModuleStandardInterface.q_dwModuleType <> 15000
        OnMouseClick:  AssignExpr=i_sZoomToExampleLeafModule, Assign=VIS_ExampleLeafModule, Type=Assignment
    Button (98,68 90x42), "Unwinder Module", invisible if: SR_VisControl.vpq_stCurrentModuleStandardInterface.q_dwModuleType <> 7
    Button (188,68 90x42), "Infeed Module", invisible if: SR_VisControl.vpq_stCurrentModuleStandardInterface.q_dwModuleType <> 5
    Button (278,68 90x42), "Crank Module", invisible if: SR_VisControl.vpq_stCurrentModuleStandardInterface.q_dwModuleType <> 11
        OnMouseClick:  Assign=VIS_CrankModule, Type=Assignment
    Button (98,110 90x42), "Sealing Module", invisible if: SR_VisControl.vpq_stCurrentModuleStandardInterface.q_dwModuleType <> 8
END_VISUALIZATION

// LMC_PacDrive/Application/VIS_AxisModule
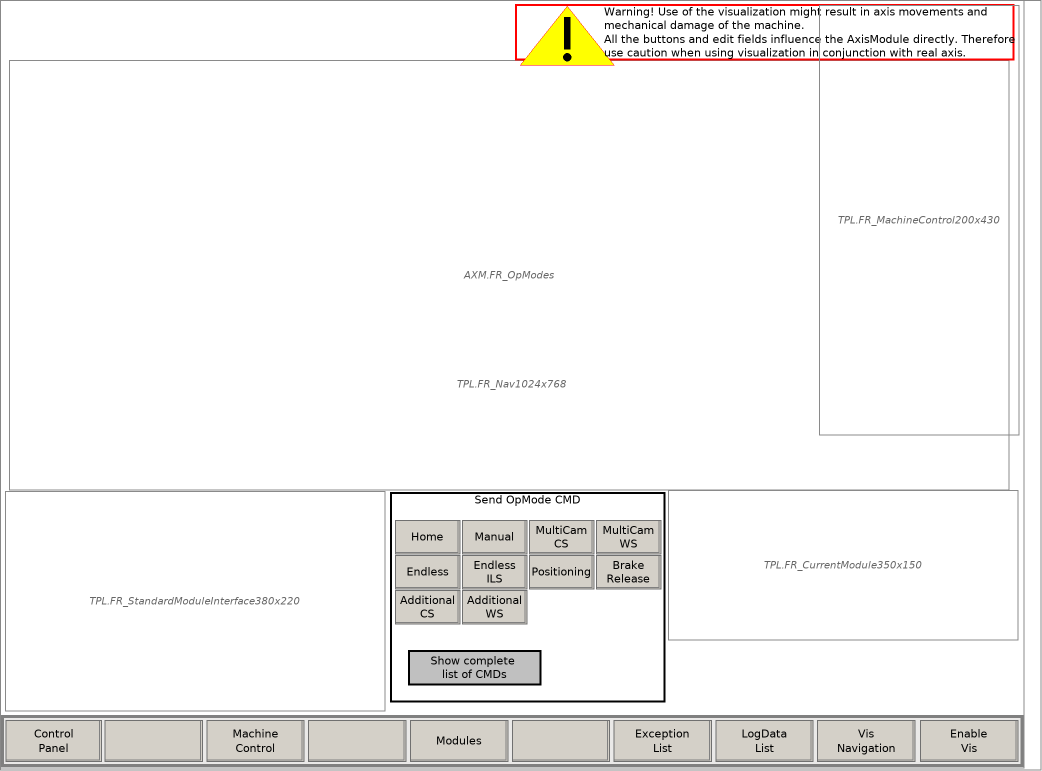
VISUALIZATION VIS_AxisModule  // 1042x771
    Frame (0,0 1024x768)
        shows TPL.FR_Nav1024x768(i_sTitle := 'Template: AxisModule')
    Frame (9,60 1000x430)
        shows AXM.FR_OpModes(iq_fbAxisModuleVisController := SR_VisControl.vpiq_fbAxisModuleVisController)
    Frame (5,491 380x220)
        shows TPL.FR_StandardModuleInterface380x220(i_stCurrentModuleStandardItf := SR_VisControl.vpq_stCurrentModuleStandardInterface, i_sCurrentModuleReaction := SR_VisControl.vpq_sCurrentModuleReaction, i_udiModuleReactionIndexMin := SR_VisControl.vpq_udiModuleReactionIndexMin, i_axModuleReaction := SR_VisControl.vpq_axModuleReaction, i_udiNumberOfReactions := SR_VisControl.udiCount, iq_xModuleReactionDown := SR_VisControl.vpiq_xModuleReactionDown, iq_xModuleReactionUp := SR_VisControl.vpiq_xModuleReactionUp, iq_diStartStepToSet := SR_VisControl.vpiq_diStartStepToSet, iq_diCmdToSet := SR_VisControl.vpiq_diCmdToSet, iq_xEnableModuleClicked := SR_VisControl.vpiq_xEnableModuleClicked, iq_xSetCmdClicked := SR_VisControl.vpiq_xSetCmdClicked, iq_fbVisContExHandling := SR_VisControl.vpiq_fbVisContExHandling)
    Rectangle (390,492 275x210), "Send OpMode CMD"
    Button (395,520 65x34), "Home", tooltip "Send CMD: ---------------------------------------------------------------- astSubModuleInterface[...].iq_diCMD := AXM.ET_Cmd.Homing (= 10);", colour toggle: SR_VisControl.v_xHomeModeActive, input disabled if: SR_VisControl.vpiq_fbAxisModuleVisController.i_pstCurrentStandardItf = 0
        OnMouseClick: execute { SR_VisControl.vpiq_fbAxisModuleVisController.i_pstCurrentStandardItf^.iq_diCmd := AXM.ET_Cmd.Homing; }
    Button (462,520 65x34), "Manual", tooltip "Send CMD: ---------------------------------------------------------------- astSubModuleInterface[...].iq_diCMD := AXM.ET_Cmd.Manual (= 20);", colour toggle: SR_VisControl.v_xManualModeActive, input disabled if: SR_VisControl.vpiq_fbAxisModuleVisController.i_pstCurrentStandardItf = 0
        OnMouseClick: execute { SR_VisControl.vpiq_fbAxisModuleVisController.i_pstCurrentStandardItf^.iq_diCmd := AXM.ET_Cmd.Manual; }
    Button (529,520 65x34), "MultiCam CS", tooltip "Send CMD: ---------------------------------------------------------------- astSubModuleInterface[...].iq_diCMD := AXM.ET_Cmd.CamCs (= 30);", colour toggle: SR_VisControl.v_xMultiCamCSActive, input disabled if: SR_VisControl.vpiq_fbAxisModuleVisController.i_pstCurrentStandardItf = 0
        OnMouseClick: execute { SR_VisControl.vpiq_fbAxisModuleVisController.i_pstCurrentStandardItf^.iq_diCmd := AXM.ET_Cmd.CamCs; }
    Button (596,520 65x34), "MultiCam WS", tooltip "Send CMD: ---------------------------------------------------------------- astSubModuleInterface[...].iq_diCMD := AXM.ET_Cmd.CamWs (= 31);", colour toggle: SR_VisControl.v_xMultiCamWSActive, input disabled if: SR_VisControl.vpiq_fbAxisModuleVisController.i_pstCurrentStandardItf = 0
        OnMouseClick: execute { SR_VisControl.vpiq_fbAxisModuleVisController.i_pstCurrentStandardItf^.iq_diCmd := AXM.ET_Cmd.CamWs; }
    Button (395,555 65x34), "Endless", tooltip "Send CMD: ---------------------------------------------------------------- astSubModuleInterface[...].iq_diCMD := AXM.ET_Cmd.Endless (= 40);", colour toggle: SR_VisControl.v_xEndlessActive, input disabled if: SR_VisControl.vpiq_fbAxisModuleVisController.i_pstCurrentStandardItf = 0
        OnMouseClick: execute { SR_VisControl.vpiq_fbAxisModuleVisController.i_pstCurrentStandardItf^.iq_diCmd := AXM.ET_Cmd.Endless; }
    Button (462,555 65x34), "Endless ILS", tooltip "Send CMD: ---------------------------------------------------------------- astSubModuleInterface[...].iq_diCMD := AXM.ET_Cmd.EndlessIls (= 41);", colour toggle: SR_VisControl.v_xEndlessILSActive, input disabled if: SR_VisControl.vpiq_fbAxisModuleVisController.i_pstCurrentStandardItf = 0
        OnMouseClick: execute { SR_VisControl.vpiq_fbAxisModuleVisController.i_pstCurrentStandardItf^.iq_diCmd := AXM.ET_Cmd.EndlessIls; }
    Button (529,555 65x34), "Positioning", tooltip "Send CMD: ---------------------------------------------------------------- astSubModuleInterface[...].iq_diCMD := AXM.ET_Cmd.Positioning (= 50);", colour toggle: SR_VisControl.v_xPositioningActive, input disabled if: SR_VisControl.vpiq_fbAxisModuleVisController.i_pstCurrentStandardItf = 0
        OnMouseClick: execute { SR_VisControl.vpiq_fbAxisModuleVisController.i_pstCurrentStandardItf^.iq_diCmd := AXM.ET_Cmd.Positioning; }
    Button (596,555 65x34), "Brake Release", tooltip "Send CMD: ---------------------------------------------------------------- astSubModuleInterface[...].iq_diCMD := AXM.ET_Cmd.BrakeRelease (= 70);", colour toggle: SR_VisControl.v_xBrakeActive, input disabled if: SR_VisControl.vpiq_fbAxisModuleVisController.i_pstCurrentStandardItf = 0
        OnMouseClick: execute { SR_VisControl.vpiq_fbAxisModuleVisController.i_pstCurrentStandardItf^.iq_diCmd := AXM.ET_Cmd.BrakeRelease; }
    Button (395,590 65x34), "Additional CS", tooltip "Send CMD: ---------------------------------------------------------------- astSubModuleInterface[...].iq_diCMD := AXM.ET_Cmd.AdditionalCs (= 80);", colour toggle: SR_VisControl.v_xAdditionalCSActive, input disabled if: SR_VisControl.vpiq_fbAxisModuleVisController.i_pstCurrentStandardItf = 0
        OnMouseClick: execute { SR_VisControl.vpiq_fbAxisModuleVisController.i_pstCurrentStandardItf^.iq_diCmd := AXM.ET_Cmd.AdditionalCs; }
    Button (462,590 65x34), "Additional WS", tooltip "Send CMD: ---------------------------------------------------------------- astSubModuleInterface[...].iq_diCMD := AXM.ET_Cmd.AdditionalWs (= 81);", colour toggle: SR_VisControl.v_xAdditionalWSActive, input disabled if: SR_VisControl.vpiq_fbAxisModuleVisController.i_pstCurrentStandardItf = 0
        OnMouseClick: execute { SR_VisControl.vpiq_fbAxisModuleVisController.i_pstCurrentStandardItf^.iq_diCmd := AXM.ET_Cmd.AdditionalWs; }
    Group (509,5 521x59)
        Rectangle (6,-1 499x56)
        Group (7,3 82x50)
            Polygon (4,57) (51,-2) (98,57) (98,57)
            Ellipse (47,45 8x8)
            RoundedRectangle (48,9 6x32)
        Rectangle (92,25 431x32), "All the buttons and edit fields influence the AxisModule directly. Therefore use caution when using visualization in conjunction with real axis."
        Rectangle (92,-2 439x31), "Warning! Use of the visualization might result in axis movements and mechanical damage of the machine."
    Frame (668,490 350x150)
        shows TPL.FR_CurrentModule350x150(i_stCurrentModuleStandardItf := SR_VisControl.vpq_stCurrentModuleStandardInterface)
    Rectangle (408,650 133x35), "Show complete list of CMDs", tooltip "(* AxisModule command area: 1-199 *) (*Selecting OpModes of FB_AxisModule*) Homing := 10 Manual := 20 CamCs := 30 CamWs := 31 Endless := 40 EndlessIls := 41 Positioning := 50 BrakeRelease := 70 AdditionalCs := 80 AdditionalWs := 81 (*ControlSignals for the selected OpMode of FB_AxisModule*) Start := 100 StartTrig := 101 StartTrigWaitInPos := 102 Stop := 110 Hold := 120 WsStart := 150 (*De-/Activating PositionControl of the respective Drive*) DriveEnableOn := 130 DriveEnableOff := 140"
    Frame (1,715 1024x54)
        shows FR_NavigationButtons()
    Frame (819,5 200x430), invisible if: NOT SR_VisControl.vpiq_xShowControlFrame
        shows TPL.FR_MachineControl200x430(i_stMachineItf := SR_VisControl.vpq_stMachineInterface, i_xPrepareActive := G_xPrepareActive, i_xAutoActive := G_xAutoActive, i_xBrakeReleaseActive := G_xBrakeReleaseActive, i_xJogMachineActive := G_xJogMachineActive, i_xManualActive := G_xManualActive, i_xException := SR_VisControl.vpq_xMachineInException, i_dwDiagQuitColor := SR_VisControl.vpq_dwDiagQuitColor, iq_iPositionX := SR_VisControl.vpiq_iPositionX, iq_iPositionY := SR_VisControl.vpiq_iPositionY, iq_xEmergencyEpas := G_xEmergencyEpas, iq_xStartEpas := G_xStartEpas, iq_xStopEpas := G_xStopEpas, iq_xJogForwEpas := G_xJogForwEpas, iq_xJogBackEpas := G_xJogBackEpas, iq_xDoPrepare := G_xDoPrepare, iq_xDoAuto := G_xDoAuto, iq_xDoBrakeRelease := G_xDoBrakeRelease, iq_xDoJogMachine := G_xDoJogMachine, iq_xDoManual := G_xDoManual, iq_xDiagQuitEpas := G_xDiagQuitEpas)
        p1457045297: SR_VisControl.stMachineInterface.stQ.xError
        p1941967854: g_I_xEmergency_Epas
        p2531571229: g_I_xStart_Epas
        p1511842254: g_I_xStop_Epas
        p745511063: g_I_xJogForw_Epas
        p3518271027: g_I_xJogBack_Epas
        p1982879521: g_I_xErrorQuit_Epas
        p3866886353: SR_VisControl.dwErrorQuitColor
        p1761348311: SR_VisControl.vpq_stMachineInterface
        p3560616238: SR_VisControl.vpiq_iPositionX
        p2738717112: SR_VisControl.vpiq_iPositionY
END_VISUALIZATION

// LMC_PacDrive/Application/VIS_ControlModule
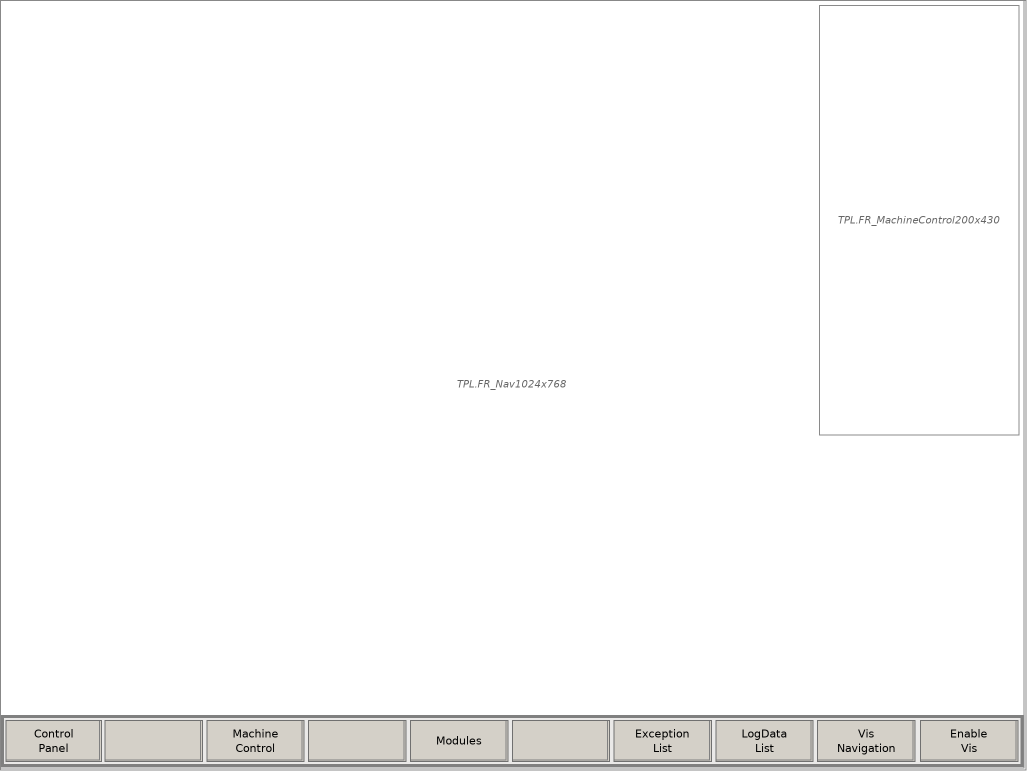
VISUALIZATION VIS_ControlModule  // 1027x771
    Frame (0,0 1024x768)
        shows TPL.FR_Nav1024x768(i_sTitle := 'Template: ControlModule')
    Frame (1,715 1024x54)
        shows FR_NavigationButtons()
    Frame (819,5 200x430), invisible if: NOT SR_VisControl.vpiq_xShowControlFrame
        shows TPL.FR_MachineControl200x430(i_stMachineItf := SR_VisControl.vpq_stMachineInterface, i_xPrepareActive := G_xPrepareActive, i_xAutoActive := G_xAutoActive, i_xBrakeReleaseActive := G_xBrakeReleaseActive, i_xJogMachineActive := G_xJogMachineActive, i_xManualActive := G_xManualActive, i_xException := SR_VisControl.vpq_xMachineInException, i_dwDiagQuitColor := SR_VisControl.vpq_dwDiagQuitColor, iq_iPositionX := SR_VisControl.vpiq_iPositionX, iq_iPositionY := SR_VisControl.vpiq_iPositionY, iq_xEmergencyEpas := G_xEmergencyEpas, iq_xStartEpas := G_xStartEpas, iq_xStopEpas := G_xStopEpas, iq_xJogForwEpas := G_xJogForwEpas, iq_xJogBackEpas := G_xJogBackEpas, iq_xDoPrepare := G_xDoPrepare, iq_xDoAuto := G_xDoAuto, iq_xDoBrakeRelease := G_xDoBrakeRelease, iq_xDoJogMachine := G_xDoJogMachine, iq_xDoManual := G_xDoManual, iq_xDiagQuitEpas := G_xDiagQuitEpas)
        p1457045297: SR_VisControl.stMachineInterface.stQ.xError
        p1941967854: g_I_xEmergency_Epas
        p2531571229: g_I_xStart_Epas
        p1511842254: g_I_xStop_Epas
        p745511063: g_I_xJogForw_Epas
        p3518271027: g_I_xJogBack_Epas
        p1982879521: g_I_xErrorQuit_Epas
        p3866886353: SR_VisControl.dwErrorQuitColor
        p1761348311: SR_VisControl.vpq_stMachineInterface
        p3560616238: SR_VisControl.vpiq_iPositionX
        p2738717112: SR_VisControl.vpiq_iPositionY
END_VISUALIZATION

// LMC_PacDrive/Application/VIS_ExceptionDetails
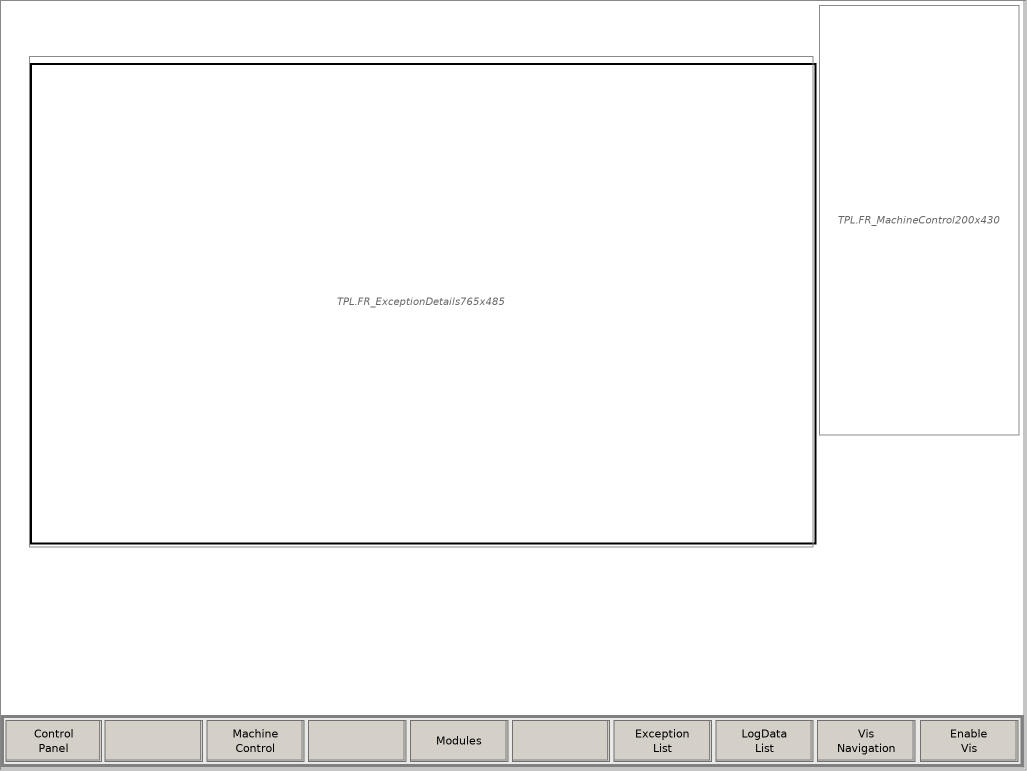
VISUALIZATION VIS_ExceptionDetails  // 1027x771
    Frame (0,0 1024x768)
        shows TPL.FR_Nav1024x768(i_sTitle := 'Template: ExceptionDetails')
    Frame (1,715 1024x54)
        shows FR_NavigationButtons()
    Rectangle (30,63 786x481)
    Frame (29,56 784x491)
        shows TPL.FR_ExceptionDetails765x485(iq_fbVisContExHandling := SR_VisControl.vpiq_fbVisContExHandling)
        p2566176161: 'Vis_ModuleErrors'
        p1989587566: 'Vis_Modules'
    Frame (819,5 200x430), invisible if: NOT SR_VisControl.vpiq_xShowControlFrame
        shows TPL.FR_MachineControl200x430(i_stMachineItf := SR_VisControl.vpq_stMachineInterface, i_xPrepareActive := G_xPrepareActive, i_xAutoActive := G_xAutoActive, i_xBrakeReleaseActive := G_xBrakeReleaseActive, i_xJogMachineActive := G_xJogMachineActive, i_xManualActive := G_xManualActive, i_xException := SR_VisControl.vpq_xMachineInException, i_dwDiagQuitColor := SR_VisControl.vpq_dwDiagQuitColor, iq_iPositionX := SR_VisControl.vpiq_iPositionX, iq_iPositionY := SR_VisControl.vpiq_iPositionY, iq_xEmergencyEpas := G_xEmergencyEpas, iq_xStartEpas := G_xStartEpas, iq_xStopEpas := G_xStopEpas, iq_xJogForwEpas := G_xJogForwEpas, iq_xJogBackEpas := G_xJogBackEpas, iq_xDoPrepare := G_xDoPrepare, iq_xDoAuto := G_xDoAuto, iq_xDoBrakeRelease := G_xDoBrakeRelease, iq_xDoJogMachine := G_xDoJogMachine, iq_xDoManual := G_xDoManual, iq_xDiagQuitEpas := G_xDiagQuitEpas)
        p1457045297: SR_VisControl.stMachineInterface.stQ.xError
        p1941967854: g_I_xEmergency_Epas
        p2531571229: g_I_xStart_Epas
        p1511842254: g_I_xStop_Epas
        p745511063: g_I_xJogForw_Epas
        p3518271027: g_I_xJogBack_Epas
        p1982879521: g_I_xErrorQuit_Epas
        p3866886353: SR_VisControl.dwErrorQuitColor
        p1761348311: SR_VisControl.vpq_stMachineInterface
        p3560616238: SR_VisControl.vpiq_iPositionX
        p2738717112: SR_VisControl.vpiq_iPositionY
END_VISUALIZATION

// LMC_PacDrive/Application/VIS_ExceptionList
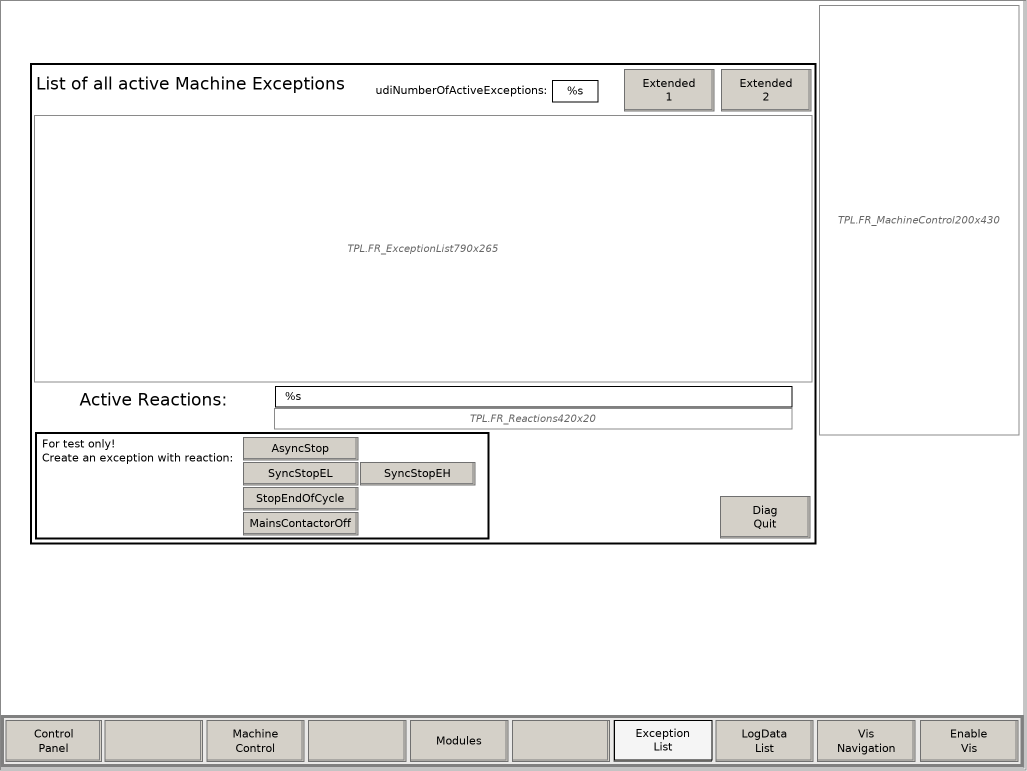
VISUALIZATION VIS_ExceptionList  // 1027x771
    Frame (0,0 1024x768)
        shows TPL.FR_Nav1024x768(i_sTitle := 'Template: ExceptionList')
    Frame (1,715 1024x54)
        shows FR_NavigationButtons()
    Rectangle (30,63 786x481)
    Rectangle (33,66 310x35), "List of all active Machine Exceptions"
    Rectangle (46,382 215x35), "Active Reactions:"
    Rectangle (369,78 181x25), "udiNumberOfActiveExceptions:"
    Rectangle (275,386 517x21), "%s", text variable: SR_VisControl.vpq_sAllActiveReactions
    Rectangle (35,432 454x107)
    Rectangle (39,436 195x29), "For test only! Create an exception with reaction:"
    Frame (274,408 518x21)
        shows TPL.FR_Reactions420x20(i_udiIndexMin := SR_VisControl.vpq_udiReactionIndexMin, i_axReaction := SR_VisControl.vpq_axReaction, i_udiNumberOfReactions := TPL.Gc_udiMaxNumberOfReactions, iq_xScrollDown := SR_VisControl.vpiq_xReactionDown, iq_xScrollUp := SR_VisControl.vpiq_xReactionUp)
        p3944911060: SR_VisControl.iErrorReactionIndexMin
        p214250784: TPC_Gc_diMaxNumberOfErrorReactions
    Button (360,462 115x23), "SyncStopEH", tooltip "For testing purpose only! Create an exception with the reaction TPL.ET_Reaction.SyncStopEH. Machine reacts with "Synchronous stop". For a detailed description of this reaction search the help index for ET_Reaction.", colour toggle: SR_VisControl.vpiq_xTestUserException3
        toggle SR_VisControl.vpiq_xTestUserException3
    Button (243,437 115x23), "AsyncStop", tooltip "For testing purpose only! Create an exception with the reaction TPL.ET_Reaction.AsyncStop. Machine reacts with "Immediate asynchronous stop". For a detailed description of this reaction search the help index for ET_Reaction.", colour toggle: SR_VisControl.vpiq_xTestUserException1
        toggle SR_VisControl.vpiq_xTestUserException1
    Button (243,462 115x23), "SyncStopEL", tooltip "For testing purpose only! Create an exception with the reaction TPL.ET_Reaction.SyncStopEL. Machine reacts with "Synchronous stop with process deactivation after stop". For a detailed description of this reaction search the help index for ET_Reaction.", colour toggle: SR_VisControl.vpiq_xTestUserException2
        toggle SR_VisControl.vpiq_xTestUserException2
    Button (243,487 115x23), "StopEndOfCycle", tooltip "For testing purpose only! Create an exception with the reaction TPL.ET_Reaction.StopEndOfCycle. Machine reacts with "Stop at end of cycle". For a detailed description of this reaction search the help index for ET_Reaction.", colour toggle: SR_VisControl.vpiq_xTestUserException4
        toggle SR_VisControl.vpiq_xTestUserException4
    Button (243,512 115x23), "MainsContactorOff", tooltip "For testing purpose only! Create an exception with the reaction TPL.ET_Reaction.MainsContactorOff. Machine reacts with "Immediate deactivation of the mains contactor". For a detailed description of this reaction search the help index for ET_Reaction.", colour toggle: SR_VisControl.vpiq_xTestUserException5
        toggle SR_VisControl.vpiq_xTestUserException5
    Button (624,69 90x42), "Extended 1", colour toggle: SR_VisControl.vpq_xShowExtendedTimes
        toggle SR_VisControl.vpiq_xButtonShowExtendedTimes
    Button (721,69 90x42), "Extended 2", colour toggle: SR_VisControl.vpq_xShowExtended2
        toggle SR_VisControl.vpiq_xButtonShowExtended2
    Textfield (552,80 46x22), "%s", text variable: G_stExceptionList.udiNumberOfActiveExceptions
    Button (720,496 90x42), "Diag Quit", colour toggle: SR_VisControl.vpq_xMachineInException
        p573394764: SR_VisControl.vpq_dwDiagQuitColor
        tap G_xDiagQuitEpas
    Frame (34,115 778x267)
        shows TPL.FR_ExceptionList790x265(i_astExceptionListTable := SR_VisControl.vpq_astExceptionListTable, i_asReaction := SR_VisControl.vpq_asReaction, i_xShowExtendedTimes := SR_VisControl.vpq_xShowExtendedTimes, i_xShowExtended2 := SR_VisControl.vpq_xShowExtended2, i_xDisplayScrollDown := SR_VisControl.vpq_xDisplayScrollDown, i_udiExceptionListIndexMax := SR_VisControl.vpq_udiExceptionListIndexMax, i_udiNumberOfExceptions := SR_VisControl.vpq_udiNumberOfExceptions, iq_udiExceptionListIndexMin := SR_VisControl.vpiq_udiExceptionListIndexMin, iq_udiExceptionListGoToDetailsOfLine := SR_VisControl.vpiq_udiExceptionListGoToDetailsOfLine)
    Rectangle (614,720 98x40), "Exception List"
    Frame (819,5 200x430), invisible if: NOT SR_VisControl.vpiq_xShowControlFrame
        shows TPL.FR_MachineControl200x430(i_stMachineItf := SR_VisControl.vpq_stMachineInterface, i_xPrepareActive := G_xPrepareActive, i_xAutoActive := G_xAutoActive, i_xBrakeReleaseActive := G_xBrakeReleaseActive, i_xJogMachineActive := G_xJogMachineActive, i_xManualActive := G_xManualActive, i_xException := SR_VisControl.vpq_xMachineInException, i_dwDiagQuitColor := SR_VisControl.vpq_dwDiagQuitColor, iq_iPositionX := SR_VisControl.vpiq_iPositionX, iq_iPositionY := SR_VisControl.vpiq_iPositionY, iq_xEmergencyEpas := G_xEmergencyEpas, iq_xStartEpas := G_xStartEpas, iq_xStopEpas := G_xStopEpas, iq_xJogForwEpas := G_xJogForwEpas, iq_xJogBackEpas := G_xJogBackEpas, iq_xDoPrepare := G_xDoPrepare, iq_xDoAuto := G_xDoAuto, iq_xDoBrakeRelease := G_xDoBrakeRelease, iq_xDoJogMachine := G_xDoJogMachine, iq_xDoManual := G_xDoManual, iq_xDiagQuitEpas := G_xDiagQuitEpas)
        p1457045297: SR_VisControl.stMachineInterface.stQ.xError
        p1941967854: g_I_xEmergency_Epas
        p2531571229: g_I_xStart_Epas
        p1511842254: g_I_xStop_Epas
        p745511063: g_I_xJogForw_Epas
        p3518271027: g_I_xJogBack_Epas
        p1982879521: g_I_xErrorQuit_Epas
        p3866886353: SR_VisControl.dwErrorQuitColor
        p1761348311: SR_VisControl.vpq_stMachineInterface
        p3560616238: SR_VisControl.vpiq_iPositionX
        p2738717112: SR_VisControl.vpiq_iPositionY
END_VISUALIZATION

// LMC_PacDrive/Application/VIS_LogDataList
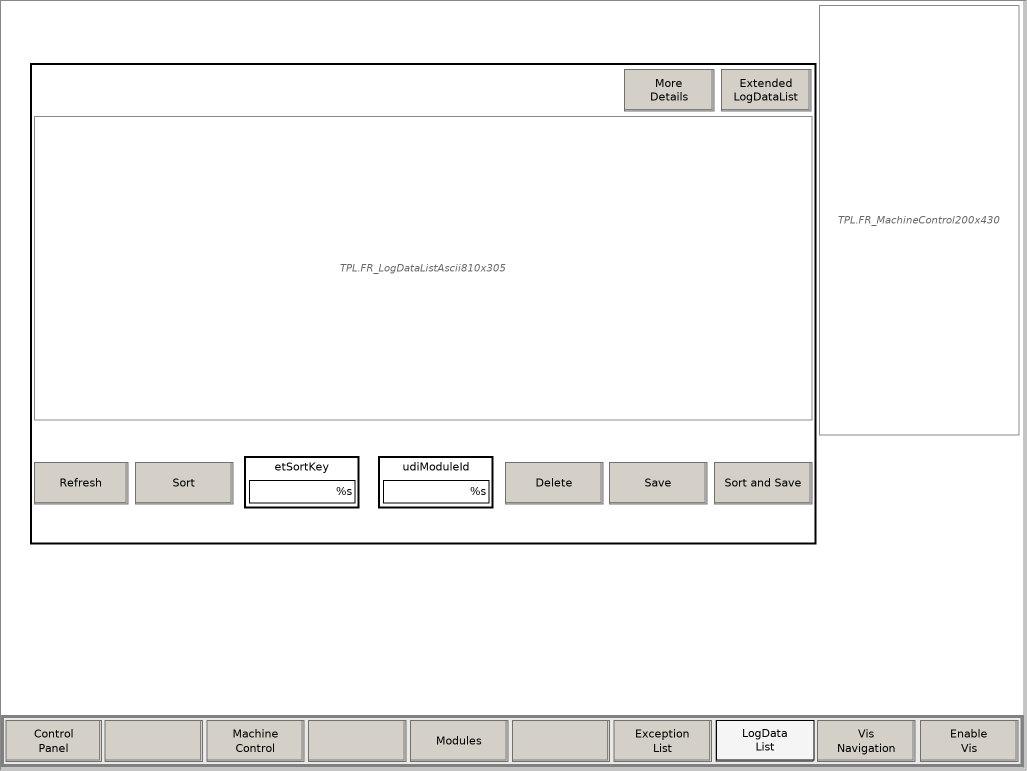
VISUALIZATION VIS_LogDataList  // 1027x771
    Frame (0,0 1024x768)
        shows TPL.FR_Nav1024x768(i_sTitle := 'Template: LogDataList')
    Frame (1,715 1024x54)
        shows FR_NavigationButtons()
    Rectangle (30,63 786x481)
    Rectangle (244,456 115x52)
    Rectangle (378,456 115x52)
    Frame (34,116 778x304)
        shows TPL.FR_LogDataListAscii810x305(i_udiLogDataListIndexMax := SR_VisControl.vpq_udiLogDataListIndexMax, i_xLogDataScrollDown := SR_VisControl.vpq_xLogDataScrollDown, i_stLogDataListAscii := G_stLogDataListAscii, i_astLogDataTable := SR_VisControl.vpq_astLogDataTable, i_xShowLogDataListDetails := SR_VisControl.vpq_xShowLogDataListDetails, iq_udiLogDataListIndexMin := SR_VisControl.vpiq_udiLogDataListIndexMin, iq_udiNumberOfLogData := SR_VisControl.vpiq_udiNumberOfLogData)
        p614390240: SR_VisControl.iLoggerListIndexMin
        p2848728500: G_stLogDataListAscii
        p1478497087: SR_VisControl.xLoggerExtendedLogger
        p3640196843: SR_VisControl.xLoggerScrollDown
        p3171618909: SR_VisControl.diNumberOfLogData
        p348598905: SR_VisControl.iLoggerListIndexMax
        p443021939: SR_VisControl.udiLoggerListIndexMax
        p1814956285: SR_VisControl.udiLoggerListIndexMin
    Button (624,69 90x42), "More Details", colour toggle: SR_VisControl.vpq_xShowLogDataListDetails
        toggle SR_VisControl.vpiq_xButtonLogDataListDetails
    Button (721,69 90x42), "Extended LogDataList"
        OnMouseClick:  Assign=VIS_LogDataListExt, Type=Assignment
    Button (135,462 98x42), "Sort", colour toggle: G_stLoggerInterface.i_xSort
        tap G_stLoggerInterface.i_xSort
    Button (34,462 94x42), "Refresh", colour toggle: G_stLoggerInterface.i_xSort
        tap G_stLoggerInterface.i_xSort
    Button (505,462 98x42), "Delete", colour toggle: G_stLoggerInterface.i_xDelete
        tap G_stLoggerInterface.i_xDelete
    Button (609,462 98x42), "Save", colour toggle: G_stLoggerInterface.i_xSave
        tap G_stLoggerInterface.i_xSave
    Button (714,462 98x42), "Sort and Save", colour toggle: G_stLoggerInterface.i_xSortAndSave
        tap G_stLoggerInterface.i_xSortAndSave
    Textfield (383,480 106x23), "%s", text variable: G_stLoggerInterface.i_udiModuleId
        OnMouseClick: write the text variable via Edit
    Textfield (249,480 106x23), "%s", tooltip "TPD_SORTBY_TIME:= 0 TPD_SORTBY_NAME:= 1 TPD_SORTBY_ID:= 2 TPD_SORTBY_CMD:= 3 TPD_SORTBY_ERRORREACTION:= 4 TPD_GE_SORTBY_MODULE_ID:= 5 TPD_GE_SORTBY_MODULE_ID_AND_TIME:= 6", text variable: G_stLoggerInterface.i_etSortKey
        OnMouseClick: write the text variable via Edit
    Rectangle (247,458 110x18), "etSortKey"
    Rectangle (381,458 110x18), "udiModuleId"
    Rectangle (716,720 98x40), "LogData List"
    Frame (819,5 200x430), invisible if: NOT SR_VisControl.vpiq_xShowControlFrame
        shows TPL.FR_MachineControl200x430(i_stMachineItf := SR_VisControl.vpq_stMachineInterface, i_xPrepareActive := G_xPrepareActive, i_xAutoActive := G_xAutoActive, i_xBrakeReleaseActive := G_xBrakeReleaseActive, i_xJogMachineActive := G_xJogMachineActive, i_xManualActive := G_xManualActive, i_xException := SR_VisControl.vpq_xMachineInException, i_dwDiagQuitColor := SR_VisControl.vpq_dwDiagQuitColor, iq_iPositionX := SR_VisControl.vpiq_iPositionX, iq_iPositionY := SR_VisControl.vpiq_iPositionY, iq_xEmergencyEpas := G_xEmergencyEpas, iq_xStartEpas := G_xStartEpas, iq_xStopEpas := G_xStopEpas, iq_xJogForwEpas := G_xJogForwEpas, iq_xJogBackEpas := G_xJogBackEpas, iq_xDoPrepare := G_xDoPrepare, iq_xDoAuto := G_xDoAuto, iq_xDoBrakeRelease := G_xDoBrakeRelease, iq_xDoJogMachine := G_xDoJogMachine, iq_xDoManual := G_xDoManual, iq_xDiagQuitEpas := G_xDiagQuitEpas)
        p1457045297: SR_VisControl.stMachineInterface.stQ.xError
        p1941967854: g_I_xEmergency_Epas
        p2531571229: g_I_xStart_Epas
        p1511842254: g_I_xStop_Epas
        p745511063: g_I_xJogForw_Epas
        p3518271027: g_I_xJogBack_Epas
        p1982879521: g_I_xErrorQuit_Epas
        p3866886353: SR_VisControl.dwErrorQuitColor
        p1761348311: SR_VisControl.vpq_stMachineInterface
        p3560616238: SR_VisControl.vpiq_iPositionX
        p2738717112: SR_VisControl.vpiq_iPositionY
END_VISUALIZATION

// LMC_PacDrive/Application/VIS_LogDataListExt
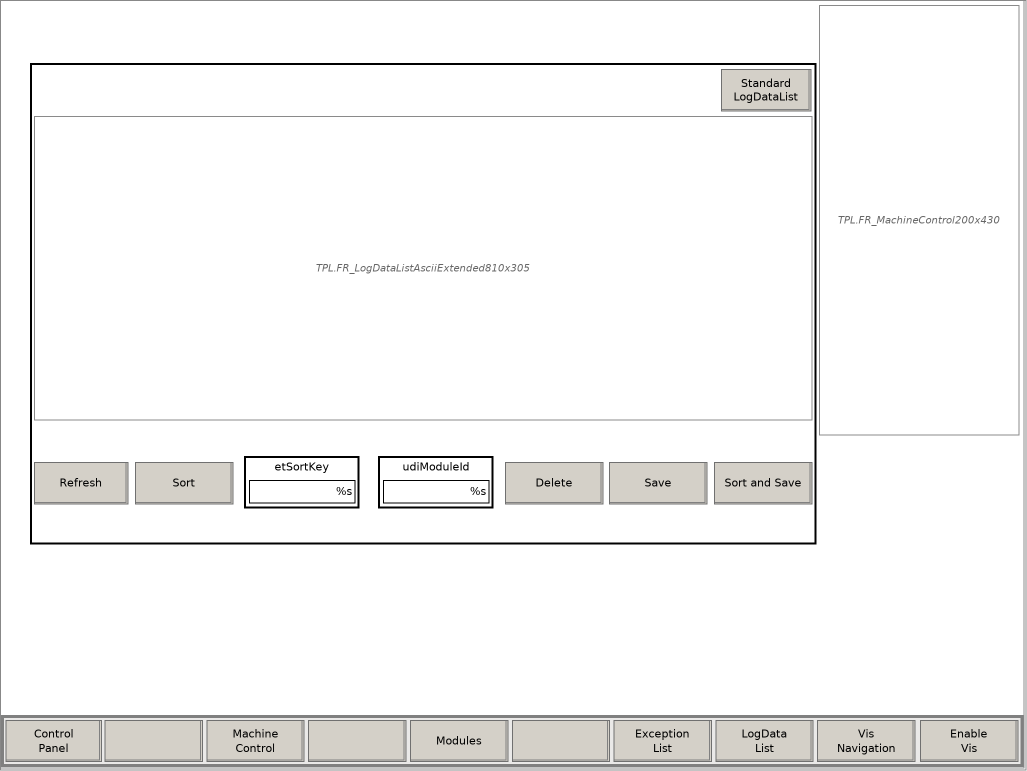
VISUALIZATION VIS_LogDataListExt  // 1027x771
    Frame (0,0 1024x768)
        shows TPL.FR_Nav1024x768(i_sTitle := 'Template: LogDataListExt')
    Frame (1,715 1024x54)
        shows FR_NavigationButtons()
    Rectangle (30,63 786x481)
    Rectangle (244,456 115x52)
    Rectangle (378,456 115x52)
    Button (135,462 98x42), "Sort", colour toggle: G_stLoggerInterface.i_xSort
        tap G_stLoggerInterface.i_xSort
    Button (34,462 94x42), "Refresh", colour toggle: G_stLoggerInterface.i_xSort
        tap G_stLoggerInterface.i_xSort
    Button (505,462 98x42), "Delete", colour toggle: G_stLoggerInterface.i_xDelete
        tap G_stLoggerInterface.i_xDelete
    Button (609,462 98x42), "Save", colour toggle: G_stLoggerInterface.i_xSave
        tap G_stLoggerInterface.i_xSave
    Button (714,462 98x42), "Sort and Save", colour toggle: G_stLoggerInterface.i_xSortAndSave
        tap G_stLoggerInterface.i_xSortAndSave
    Textfield (383,480 106x23), "%s", text variable: G_stLoggerInterface.i_udiModuleId
        OnMouseClick: write the text variable via Edit
    Textfield (249,480 106x23), "%s", tooltip "TPD_SORTBY_TIME:= 0 TPD_SORTBY_NAME:= 1 TPD_SORTBY_ID:= 2 TPD_SORTBY_CMD:= 3 TPD_SORTBY_ERRORREACTION:= 4 TPD_GE_SORTBY_MODULE_ID:= 5 TPD_GE_SORTBY_MODULE_ID_AND_TIME:= 6", text variable: G_stLoggerInterface.i_etSortKey
        OnMouseClick: write the text variable via Edit
    Rectangle (247,458 110x18), "etSortKey"
    Rectangle (381,458 110x18), "udiModuleId"
    Button (721,69 90x42), "Standard LogDataList"
        OnMouseClick:  Assign=VIS_LogDataList, Type=Assignment
    Frame (34,116 778x304)
        shows TPL.FR_LogDataListAsciiExtended810x305(i_udiLogDataListIndexMax := SR_VisControl.vpq_udiLogDataListIndexMax, i_xLogDataScrollDown := SR_VisControl.vpq_xLogDataScrollDown, i_stLogDataListAscii := G_stLogDataListAscii, i_astLogDataTable := SR_VisControl.vpq_astLogDataTable, i_astLogDataTableAscii := SR_VisControl.vpq_astLogDataTableAscii, iq_udiLogDataListIndexMin := SR_VisControl.vpiq_udiLogDataListIndexMin, iq_udiNumberOfLogData := SR_VisControl.vpiq_udiNumberOfLogData)
        p2848728500: G_stLogDataListAscii
        p3166277772: SR_VisControl.astLogDataTable
        p348598905: SR_VisControl.iLoggerListIndexMax
        p614390240: SR_VisControl.iLoggerListIndexMin
        p3640196843: SR_VisControl.xLoggerScrollDown
        p3171618909: SR_VisControl.diNumberOfLogData
        p443021939: SR_VisControl.udiLoggerListIndexMax
        p1478497087: SR_VisControl.xLoggerExtendedLogger
        p1814956285: SR_VisControl.udiLoggerListIndexMin
    Frame (819,5 200x430), invisible if: NOT SR_VisControl.vpiq_xShowControlFrame
        shows TPL.FR_MachineControl200x430(i_stMachineItf := SR_VisControl.vpq_stMachineInterface, i_xPrepareActive := G_xPrepareActive, i_xAutoActive := G_xAutoActive, i_xBrakeReleaseActive := G_xBrakeReleaseActive, i_xJogMachineActive := G_xJogMachineActive, i_xManualActive := G_xManualActive, i_xException := SR_VisControl.vpq_xMachineInException, i_dwDiagQuitColor := SR_VisControl.vpq_dwDiagQuitColor, iq_iPositionX := SR_VisControl.vpiq_iPositionX, iq_iPositionY := SR_VisControl.vpiq_iPositionY, iq_xEmergencyEpas := G_xEmergencyEpas, iq_xStartEpas := G_xStartEpas, iq_xStopEpas := G_xStopEpas, iq_xJogForwEpas := G_xJogForwEpas, iq_xJogBackEpas := G_xJogBackEpas, iq_xDoPrepare := G_xDoPrepare, iq_xDoAuto := G_xDoAuto, iq_xDoBrakeRelease := G_xDoBrakeRelease, iq_xDoJogMachine := G_xDoJogMachine, iq_xDoManual := G_xDoManual, iq_xDiagQuitEpas := G_xDiagQuitEpas)
        p1457045297: SR_VisControl.stMachineInterface.stQ.xError
        p1941967854: g_I_xEmergency_Epas
        p2531571229: g_I_xStart_Epas
        p1511842254: g_I_xStop_Epas
        p745511063: g_I_xJogForw_Epas
        p3518271027: g_I_xJogBack_Epas
        p1982879521: g_I_xErrorQuit_Epas
        p3866886353: SR_VisControl.dwErrorQuitColor
        p1761348311: SR_VisControl.vpq_stMachineInterface
        p3560616238: SR_VisControl.vpiq_iPositionX
        p2738717112: SR_VisControl.vpiq_iPositionY
END_VISUALIZATION

// LMC_PacDrive/Application/VIS_ModuleDetails
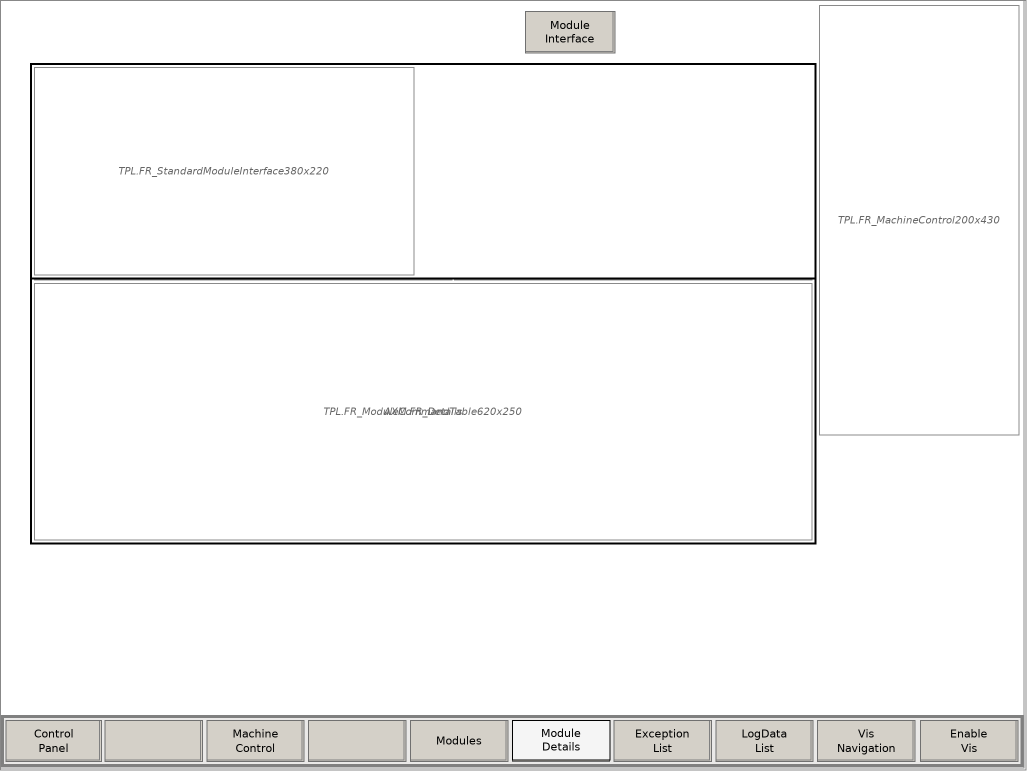
VISUALIZATION VIS_ModuleDetails  // 1027x771
    Frame (0,0 1024x768)
        shows TPL.FR_Nav1024x768(i_sTitle := 'Template: ModuleDetails')
    Frame (1,715 1024x54)
        shows FR_NavigationButtons()
    Button (525,11 90x42), "Module Interface", colour toggle: SR_VisControl.vpiq_xShowModuleInterface
        toggle SR_VisControl.vpiq_xShowModuleInterface
    Rectangle (30,63 786x481)
    Frame (34,128 418x152)
        shows TPL.FR_Navigation360x150(i_sNameNavRight := SR_VisControl.vpq_sNameNavRight, i_sNameNavUp := SR_VisControl.vpq_sNameNavUp, i_sNameNavLeft := SR_VisControl.vpq_sNameNavLeft, i_sNameNavDown := SR_VisControl.vpq_sNameNavDown, i_xEnableNavUp := SR_VisControl.vpq_xEnableNavUp, i_xEnableNavLeft := SR_VisControl.vpq_xEnableNavLeft, i_xEnableNavRight := SR_VisControl.vpq_xEnableNavRight, i_xEnableNavDown := SR_VisControl.vpq_xEnableNavDown, iq_xNavUp := SR_VisControl.vpiq_xNavUp, iq_xNavLeft := SR_VisControl.vpiq_xNavLeft, iq_xNavRight := SR_VisControl.vpiq_xNavRight, iq_xNavDown := SR_VisControl.vpiq_xNavDown)
    Rectangle (30,64 786x60)
    Button (602,65 118x29), "EQModule: %s", tooltip "%s", text variable: SR_VisControl.vpq_audiIdModuleList[5], colour toggle: SR_VisControl.vpq_axActiveModuleList[5], invisible if: SR_VisControl.vpq_axDisableModuleList[5] OR SR_VisControl.vpq_axIdModuleListValid[5] = FALSE, input disabled if: SR_VisControl.vpq_axDisableModuleList[5]
        p4168582468: SR_VisControl.vpq_asNameModuleList[5]
        toggle SR_VisControl.vpiq_axModuleList[5]
    Button (483,65 118x29), "EQModule: %s", tooltip "%s", text variable: SR_VisControl.vpq_audiIdModuleList[4], colour toggle: SR_VisControl.vpq_axActiveModuleList[4], invisible if: SR_VisControl.vpq_axDisableModuleList[4] OR SR_VisControl.vpq_axIdModuleListValid[4] = FALSE, input disabled if: SR_VisControl.vpq_axDisableModuleList[4]
        p4168582468: SR_VisControl.vpq_asNameModuleList[4]
        toggle SR_VisControl.vpiq_axModuleList[4]
    Button (365,65 118x29), "EQModule: %s", tooltip "%s", text variable: SR_VisControl.vpq_audiIdModuleList[3], colour toggle: SR_VisControl.vpq_axActiveModuleList[3], invisible if: SR_VisControl.vpq_axDisableModuleList[3] OR SR_VisControl.vpq_axIdModuleListValid[3] = FALSE, input disabled if: SR_VisControl.vpq_axDisableModuleList[3]
        p4168582468: SR_VisControl.vpq_asNameModuleList[3]
        toggle SR_VisControl.vpiq_axModuleList[3]
    Button (246,65 118x29), "EQModule: %s", tooltip "%s", text variable: SR_VisControl.vpq_audiIdModuleList[2], colour toggle: SR_VisControl.vpq_axActiveModuleList[2], invisible if: SR_VisControl.vpq_axDisableModuleList[2] OR SR_VisControl.vpq_axIdModuleListValid[2] = FALSE, input disabled if: SR_VisControl.vpq_axDisableModuleList[2]
        p4168582468: SR_VisControl.vpq_asNameModuleList[2]
        toggle SR_VisControl.vpiq_axModuleList[2]
    Button (126,65 119x29), "EQModule: %s", tooltip "%s", text variable: SR_VisControl.vpq_audiIdModuleList[1], colour toggle: SR_VisControl.vpq_axActiveModuleList[1], invisible if: SR_VisControl.vpq_axDisableModuleList[1] OR SR_VisControl.vpq_axIdModuleListValid[1] = FALSE, input disabled if: SR_VisControl.vpq_axDisableModuleList[1]
        p4168582468: SR_VisControl.vpq_asNameModuleList[1]
        toggle SR_VisControl.vpiq_axModuleList[1]
    Button (126,95 119x29), "SubEQModule: %s", tooltip "%s", text variable: SR_VisControl.vpq_audiIdSubModuleList[1], colour toggle: SR_VisControl.vpq_axActiveSubModuleList[1], invisible if: SR_VisControl.vpq_axDisableSubModuleList[1] OR SR_VisControl.vpq_axIdSubModuleListValid[1] = FALSE, input disabled if: SR_VisControl.vpq_axDisableSubModuleList[1]
        p4168582468: SR_VisControl.vpq_asNameSubModuleList[1]
        toggle SR_VisControl.vpiq_axSubModuleList[1]
    Button (246,95 118x29), "SubEQModule: %s", tooltip "%s", text variable: SR_VisControl.vpq_audiIdSubModuleList[2], colour toggle: SR_VisControl.vpq_axActiveSubModuleList[2], invisible if: SR_VisControl.vpq_axDisableSubModuleList[2] OR SR_VisControl.vpq_axIdSubModuleListValid[2] = FALSE, input disabled if: SR_VisControl.vpq_axDisableSubModuleList[2]
        p4168582468: SR_VisControl.vpq_asNameSubModuleList[2]
        toggle SR_VisControl.vpiq_axSubModuleList[2]
    Button (365,95 118x29), "SubEQModule: %s", tooltip "%s", text variable: SR_VisControl.vpq_audiIdSubModuleList[3], colour toggle: SR_VisControl.vpq_axActiveSubModuleList[3], invisible if: SR_VisControl.vpq_axDisableSubModuleList[3] OR SR_VisControl.vpq_axIdSubModuleListValid[3] = FALSE, input disabled if: SR_VisControl.vpq_axDisableSubModuleList[3]
        p4168582468: SR_VisControl.vpq_asNameSubModuleList[3]
        toggle SR_VisControl.vpiq_axSubModuleList[3]
    Button (484,95 117x29), "SubEQModule: %s", tooltip "%s", text variable: SR_VisControl.vpq_audiIdSubModuleList[4], colour toggle: SR_VisControl.vpq_axActiveSubModuleList[4], invisible if: SR_VisControl.vpq_axDisableSubModuleList[4] OR SR_VisControl.vpq_axIdSubModuleListValid[4] = FALSE, input disabled if: SR_VisControl.vpq_axDisableSubModuleList[4]
        p4168582468: SR_VisControl.vpq_asNameSubModuleList[4]
        toggle SR_VisControl.vpiq_axSubModuleList[4]
    Button (602,95 118x29), "SubEQModule: %s", tooltip "%s", text variable: SR_VisControl.vpq_audiIdSubModuleList[5], colour toggle: SR_VisControl.vpq_axActiveSubModuleList[5], invisible if: SR_VisControl.vpq_axDisableSubModuleList[5] OR SR_VisControl.vpq_axIdSubModuleListValid[5] = FALSE, input disabled if: SR_VisControl.vpq_axDisableSubModuleList[5]
        p4168582468: SR_VisControl.vpq_asNameSubModuleList[5]
        toggle SR_VisControl.vpiq_axSubModuleList[5]
    Rectangle (720,94 95x29), ">"
    Rectangle (720,64 95x30), ">"
    Button (721,65 95x29), ">", invisible if: SR_VisControl.vpq_xDisableModuleListUp, input disabled if: SR_VisControl.vpq_xDisableModuleListUp
        toggle SR_VisControl.vpiq_xModuleListUp
    Button (721,95 95x29), ">", invisible if: SR_VisControl.vpq_xDisableSubModuleListUp, input disabled if: SR_VisControl.vpq_xDisableSubModuleListUp
        toggle SR_VisControl.vpiq_xSubModuleListUp
    Rectangle (31,94 94x29), "<"
    Rectangle (31,64 94x30), "<"
    Button (32,65 93x29), "<", invisible if: SR_VisControl.vpq_xDisableModuleListDown, input disabled if: SR_VisControl.vpq_xDisableModuleListDown
        toggle SR_VisControl.vpiq_xModuleListDown
    Button (32,95 93x29), "<", invisible if: SR_VisControl.vpq_xDisableSubModuleListDown, input disabled if: SR_VisControl.vpq_xDisableSubModuleListDown
        toggle SR_VisControl.vpiq_xSubModuleListDown
    Button (126,65 119x29), "CtrlModule: %s", tooltip "%s", text variable: SR_VisControl.vpq_asControlModuleButtonName[1], colour toggle: SR_VisControl.vpq_axControlModuleActive[1], invisible if: SR_VisControl.vpq_axControlModuleValid[1]=FALSE
        p4168582468: SR_VisControl.vpq_asToolTipControlModuleList[1]
        toggle SR_VisControl.vpiq_axControlModuleList[1]
    Button (246,65 118x29), "CtrlModule: %s", tooltip "%s", text variable: SR_VisControl.vpq_asControlModuleButtonName[2], colour toggle: SR_VisControl.vpq_axControlModuleActive[2], invisible if: SR_VisControl.vpq_axControlModuleValid[2]=FALSE
        p4168582468: SR_VisControl.vpq_asToolTipControlModuleList[2]
        toggle SR_VisControl.vpiq_axControlModuleList[2]
    Button (365,65 118x29), "CtrlModule: %s", tooltip "%s", text variable: SR_VisControl.vpq_asControlModuleButtonName[3], colour toggle: SR_VisControl.vpq_axControlModuleActive[3], invisible if: SR_VisControl.vpq_axControlModuleValid[3]=FALSE
        p4168582468: SR_VisControl.vpq_asToolTipControlModuleList[3]
        toggle SR_VisControl.vpiq_axControlModuleList[3]
    Button (484,65 117x29), "CtrlModule: %s", tooltip "%s", text variable: SR_VisControl.vpq_asControlModuleButtonName[4], colour toggle: SR_VisControl.vpq_axControlModuleActive[4], invisible if: SR_VisControl.vpq_axControlModuleValid[4]=FALSE
        p4168582468: SR_VisControl.vpq_asToolTipControlModuleList[4]
        toggle SR_VisControl.vpiq_axControlModuleList[4]
    Button (602,65 118x29), "CtrlModule: %s", tooltip "%s", text variable: SR_VisControl.vpq_asControlModuleButtonName[5], colour toggle: SR_VisControl.vpq_axControlModuleActive[5], invisible if: SR_VisControl.vpq_axControlModuleValid[5]=FALSE
        p4168582468: SR_VisControl.vpq_asToolTipControlModuleList[5]
        toggle SR_VisControl.vpiq_axControlModuleList[5]
    Button (126,95 119x29), "SubCtrlModule: %s", tooltip "%s", text variable: SR_VisControl.vpq_asSubControlModuleButtonName[1], colour toggle: SR_VisControl.vpq_axSubControlModuleActive[1], invisible if: SR_VisControl.vpq_axSubControlModuleValid[1]=FALSE
        p4168582468: SR_VisControl.vpq_asToolTipSubControlModuleList[1]
        toggle SR_VisControl.vpiq_axSubControlModuleList[1]
    Button (246,95 118x29), "SubCtrlModule: %s", tooltip "%s", text variable: SR_VisControl.vpq_asSubControlModuleButtonName[2], colour toggle: SR_VisControl.vpq_axSubControlModuleActive[2], invisible if: SR_VisControl.vpq_axSubControlModuleValid[2]=FALSE
        p4168582468: SR_VisControl.vpq_asToolTipSubControlModuleList[2]
        toggle SR_VisControl.vpiq_axSubControlModuleList[2]
    Button (365,95 118x29), "SubCtrlModule: %s", tooltip "%s", text variable: SR_VisControl.vpq_asSubControlModuleButtonName[3], colour toggle: SR_VisControl.vpq_axSubControlModuleActive[3], invisible if: SR_VisControl.vpq_axSubControlModuleValid[3]=FALSE
        p4168582468: SR_VisControl.vpq_asToolTipSubControlModuleList[3]
        toggle SR_VisControl.vpiq_axSubControlModuleList[3]
    Button (484,95 117x29), "SubCtrlModule: %s", tooltip "%s", text variable: SR_VisControl.vpq_asSubControlModuleButtonName[4], colour toggle: SR_VisControl.vpq_axSubControlModuleActive[4], invisible if: SR_VisControl.vpq_axSubControlModuleValid[4]=FALSE
        p4168582468: SR_VisControl.vpq_asToolTipSubControlModuleList[4]
        toggle SR_VisControl.vpiq_axSubControlModuleList[4]
    Button (602,95 118x29), "SubCtrlModule: %s", tooltip "%s", text variable: SR_VisControl.vpq_asSubControlModuleButtonName[5], colour toggle: SR_VisControl.vpq_axSubControlModuleActive[5], invisible if: SR_VisControl.vpq_axSubControlModuleValid[5]=FALSE
        p4168582468: SR_VisControl.vpq_asToolTipSubControlModuleList[5]
        toggle SR_VisControl.vpiq_axSubControlModuleList[5]
    Frame (454,127 358x153)
        shows TPL.FR_CurrentModule350x150(i_stCurrentModuleStandardItf := SR_VisControl.vpq_stCurrentModuleStandardInterface)
        p2332068554: SR_VisControl.stCurrentModuleStandardInterface
        p427866952: SR_VisControl.stCurrentModuleStandardInterface
        p2190627833: SR_VisControl.vpq_stCurrentModuleStandardInterface
    Rectangle (30,63 786x216), invisible if: NOT SR_VisControl.vpiq_xShowModuleInterface
    Frame (34,67 380x208), invisible if: NOT SR_VisControl.vpiq_xShowModuleInterface
        shows TPL.FR_StandardModuleInterface380x220(i_stCurrentModuleStandardItf := SR_VisControl.vpq_stCurrentModuleStandardInterface, i_sCurrentModuleReaction := SR_VisControl.vpq_sCurrentModuleReaction, i_udiModuleReactionIndexMin := SR_VisControl.vpq_udiModuleReactionIndexMin, i_axModuleReaction := SR_VisControl.vpq_axModuleReaction, i_udiNumberOfReactions := TPL.Gc_udiMaxNumberOfReactions, iq_xModuleReactionDown := SR_VisControl.vpiq_xModuleReactionDown, iq_xModuleReactionUp := SR_VisControl.vpiq_xModuleReactionUp, iq_diStartStepToSet := SR_VisControl.vpiq_diStartStepToSet, iq_diCmdToSet := SR_VisControl.vpiq_diCmdToSet, iq_xEnableModuleClicked := SR_VisControl.vpiq_xEnableModuleClicked, iq_xSetCmdClicked := SR_VisControl.vpiq_xSetCmdClicked, iq_fbVisContExHandling := SR_VisControl.vpiq_fbVisContExHandling)
        p1094400588: SR_VisControl.IFB_AxisModuleVisController.xCurrentIsOfMyType
        p3339340907: ''
        p1029787830: SR_VisControl.fbVisContExHandling
        p2258115317: SR_VisControl.iModuleErrorReactionIndexMin
        p2777435286: SR_VisControl.axModuleErrorReaction
        p214250784: TPC_Gc_diMaxNumberOfErrorReactions
        p311732222: SR_VisControl.stCurrentModuleStandardInterface
        p640132070: SR_VisControl.xModuleErrorReactionDown
        p4234372197: SR_VisControl.xModuleErrorReactionUp
        p2938682392: SR_VisControl.xEnableModule_Clicked
        p3592490199: SR_VisControl.xSetCmd_Clicked
        p2307280719: SR_VisControl.stCurrentModuleStandardInterface
        p2190627833: SR_VisControl.vpq_stCurrentModuleStandardInterface
    Frame (34,283 778x257), invisible if: SR_VisControl.vpq_stCurrentModuleStandardInterface.q_dwModuleType <> 3
        shows AXM.FR_Details(iq_fbAxisModuleVisController := SR_VisControl.vpiq_fbAxisModuleVisController)
        p334560860: SR_VisControl.IFB_AxisModuleVisController.stCurrentAxisInterface
        p159172089: SR_VisControl.IFB_AxisModuleVisController
        p2012682765: SR_VisControl.stCurrentModuleStandardInterface
        p3545344757: SR_VisControl.stCurrentModuleStandardInterface.i_sModuleName
        p2977392050: SR_VisControl.astEQCMDTable
        p1710090269: SR_VisControl.udiEQTableStepCount
        p3492251336: SR_VisControl.stCurrentModuleStandardInterface.iq_stExt.diActiveStep
        p1862340509: SR_VisControl.sEQCMDTableTitle
        p577637124: SR_VisControl.xDoEnable
        p706691565: NOT SR_VisControl.xEnableCmdTableUp
        p2658775966: NOT SR_VisControl.xEnableCmdTableDown
        p2041874301: SR_VisControl.udiEQTableIndexMin
        p427866952: SR_VisControl.stCurrentModuleStandardInterface
        p4226816124: SR_VisControl.udiEQTableIndexMin
        p2190627833: SR_VisControl.stCurrentModuleStandardInterface
    Frame (34,283 778x257), invisible if: NOT SR_VisControl.vpq_xDisplayCmdTable
        shows TPL.FR_ModuleCommandTable620x250(i_stCurrentModuleStandardItf := SR_VisControl.vpq_stCurrentModuleStandardInterface, i_astActualCmdTable := SR_VisControl.vpq_astActualCmdTableModule, i_udiNumberOfCmdSteps := SR_VisControl.vpq_udiNumberOfCmdStepsModule, i_sCmdTitel := SR_VisControl.vpq_sCmdTitleModule, i_xDoEnable := SR_VisControl.vpq_xDoEnable, i_xDisableScrollUp := SR_VisControl.vpq_xDisableScrollUpModule, i_xDisableScrollDown := SR_VisControl.vpq_xDisableScrollDownModule, iq_udiIndexMin := SR_VisControl.vpiq_udiIndexMinModule)
        p334560860: SR_VisControl.IFB_AxisModuleVisController.stCurrentAxisInterface
        p159172089: SR_VisControl.IFB_AxisModuleVisController
        p2012682765: SR_VisControl.stCurrentModuleStandardInterface
        p3545344757: SR_VisControl.stCurrentModuleStandardInterface.i_sModuleName
        p3492251336: SR_VisControl.vpq_stCurrentModuleStandardInterface.iq_stExt.diActiveStep
        p2041874301: SR_VisControl.udiEQTableIndexMin
        p427866952: SR_VisControl.stCurrentModuleStandardInterface
        p2190627833: SR_VisControl.vpq_stCurrentModuleStandardInterface
    Frame (819,5 200x430), invisible if: NOT SR_VisControl.vpiq_xShowControlFrame
        shows TPL.FR_MachineControl200x430(i_stMachineItf := SR_VisControl.vpq_stMachineInterface, i_xPrepareActive := G_xPrepareActive, i_xAutoActive := G_xAutoActive, i_xBrakeReleaseActive := G_xBrakeReleaseActive, i_xJogMachineActive := G_xJogMachineActive, i_xManualActive := G_xManualActive, i_xException := SR_VisControl.vpq_xMachineInException, i_dwDiagQuitColor := SR_VisControl.vpq_dwDiagQuitColor, iq_iPositionX := SR_VisControl.vpiq_iPositionX, iq_iPositionY := SR_VisControl.vpiq_iPositionY, iq_xEmergencyEpas := G_xEmergencyEpas, iq_xStartEpas := G_xStartEpas, iq_xStopEpas := G_xStopEpas, iq_xJogForwEpas := G_xJogForwEpas, iq_xJogBackEpas := G_xJogBackEpas, iq_xDoPrepare := G_xDoPrepare, iq_xDoAuto := G_xDoAuto, iq_xDoBrakeRelease := G_xDoBrakeRelease, iq_xDoJogMachine := G_xDoJogMachine, iq_xDoManual := G_xDoManual, iq_xDiagQuitEpas := G_xDiagQuitEpas)
        p1457045297: SR_VisControl.stMachineInterface.stQ.xError
        p1941967854: g_I_xEmergency_Epas
        p2531571229: g_I_xStart_Epas
        p1511842254: g_I_xStop_Epas
        p745511063: g_I_xJogForw_Epas
        p3518271027: g_I_xJogBack_Epas
        p1982879521: g_I_xErrorQuit_Epas
        p3866886353: SR_VisControl.dwErrorQuitColor
        p1761348311: SR_VisControl.vpq_stMachineInterface
        p3560616238: SR_VisControl.vpiq_iPositionX
        p2738717112: SR_VisControl.vpiq_iPositionY
    Rectangle (512,720 98x40), "Module Details"
END_VISUALIZATION

// LMC_PacDrive/Application/VIS_ModuleExceptions
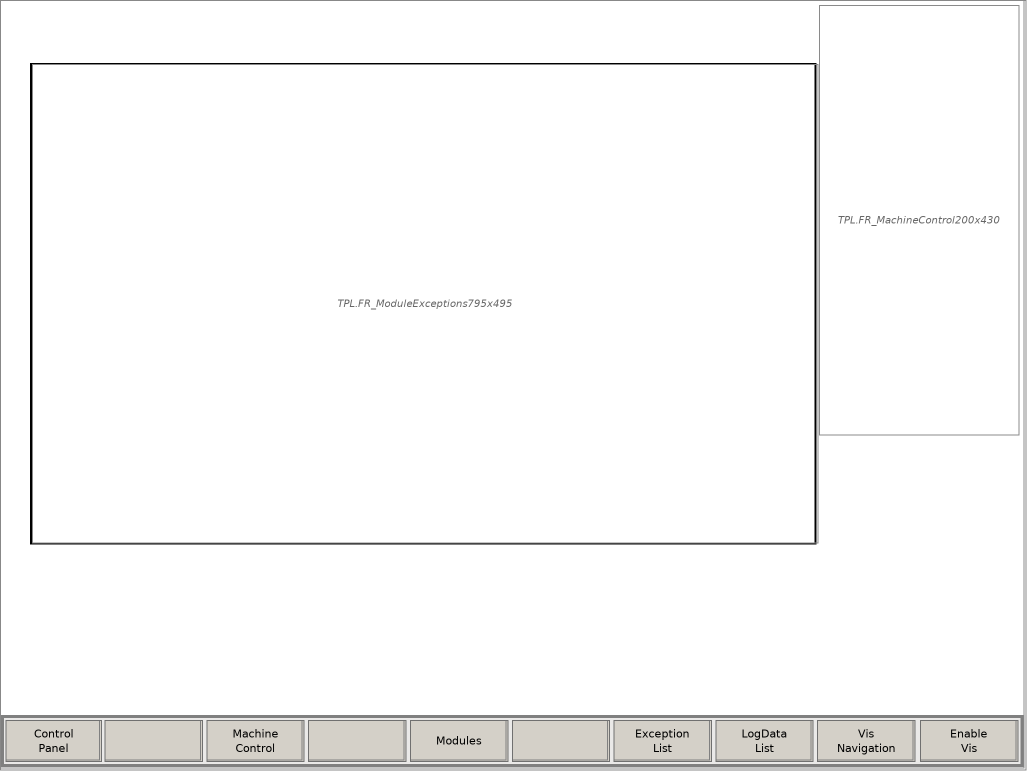
VISUALIZATION VIS_ModuleExceptions  // 1027x771
    Frame (0,0 1024x768)
        shows TPL.FR_Nav1024x768(i_sTitle := 'Template: ModuleExceptions')
    Rectangle (30,63 786x481)
    Frame (32,64 786x479)
        shows TPL.FR_ModuleExceptions795x495(i_stCurrentModuleStandardItf := SR_VisControl.vpq_stCurrentModuleStandardInterface, i_sCurrentModuleReaction := SR_VisControl.vpq_sCurrentModuleReaction, i_udiModuleReactionIndexMin := SR_VisControl.vpq_udiModuleReactionIndexMin, i_axModuleReaction := SR_VisControl.vpq_axModuleReaction, i_udiNumberOfReactions := TPL.Gc_udiMaxNumberOfReactions, iq_xModuleReactionDown := SR_VisControl.vpiq_xModuleReactionDown, iq_xModuleReactionUp := SR_VisControl.vpiq_xModuleReactionUp, iq_diStartStepToSet := SR_VisControl.vpiq_diStartStepToSet, iq_diCmdToSet := SR_VisControl.vpiq_diCmdToSet, iq_xEnableModuleClicked := SR_VisControl.vpiq_xEnableModuleClicked, iq_xSetCmdClicked := SR_VisControl.vpiq_xSetCmdClicked, iq_fbVisContExHandling := SR_VisControl.vpiq_fbVisContExHandling)
        p1094400588: SR_VisControl.IFB_AxisModuleVisController.xCurrentIsOfMyType
        p2258115317: SR_VisControl.iModuleErrorReactionIndexMin
        p2777435286: SR_VisControl.axModuleErrorReaction
        p214250784: TPC_Gc_diMaxNumberOfErrorReactions
        p311732222: SR_VisControl.stCurrentModuleStandardInterface
        p640132070: SR_VisControl.xModuleErrorReactionDown
        p4234372197: SR_VisControl.xModuleErrorReactionUp
        p2938682392: SR_VisControl.xEnableModule_Clicked
        p3592490199: SR_VisControl.xSetCmd_Clicked
        p2307280719: SR_VisControl.stCurrentModuleStandardInterface
        p2190627833: SR_VisControl.vpq_stCurrentModuleStandardInterface
    Frame (1,715 1024x54)
        shows FR_NavigationButtons()
    Frame (819,5 200x430), invisible if: NOT SR_VisControl.vpiq_xShowControlFrame
        shows TPL.FR_MachineControl200x430(i_stMachineItf := SR_VisControl.vpq_stMachineInterface, i_xPrepareActive := G_xPrepareActive, i_xAutoActive := G_xAutoActive, i_xBrakeReleaseActive := G_xBrakeReleaseActive, i_xJogMachineActive := G_xJogMachineActive, i_xManualActive := G_xManualActive, i_xException := SR_VisControl.vpq_xMachineInException, i_dwDiagQuitColor := SR_VisControl.vpq_dwDiagQuitColor, iq_iPositionX := SR_VisControl.vpiq_iPositionX, iq_iPositionY := SR_VisControl.vpiq_iPositionY, iq_xEmergencyEpas := G_xEmergencyEpas, iq_xStartEpas := G_xStartEpas, iq_xStopEpas := G_xStopEpas, iq_xJogForwEpas := G_xJogForwEpas, iq_xJogBackEpas := G_xJogBackEpas, iq_xDoPrepare := G_xDoPrepare, iq_xDoAuto := G_xDoAuto, iq_xDoBrakeRelease := G_xDoBrakeRelease, iq_xDoJogMachine := G_xDoJogMachine, iq_xDoManual := G_xDoManual, iq_xDiagQuitEpas := G_xDiagQuitEpas)
        p1457045297: SR_VisControl.stMachineInterface.stQ.xError
        p1941967854: g_I_xEmergency_Epas
        p2531571229: g_I_xStart_Epas
        p1511842254: g_I_xStop_Epas
        p745511063: g_I_xJogForw_Epas
        p3518271027: g_I_xJogBack_Epas
        p1982879521: g_I_xErrorQuit_Epas
        p3866886353: SR_VisControl.dwErrorQuitColor
        p1761348311: SR_VisControl.vpq_stMachineInterface
        p3560616238: SR_VisControl.vpiq_iPositionX
        p2738717112: SR_VisControl.vpiq_iPositionY
END_VISUALIZATION

// LMC_PacDrive/Application/VIS_Modules
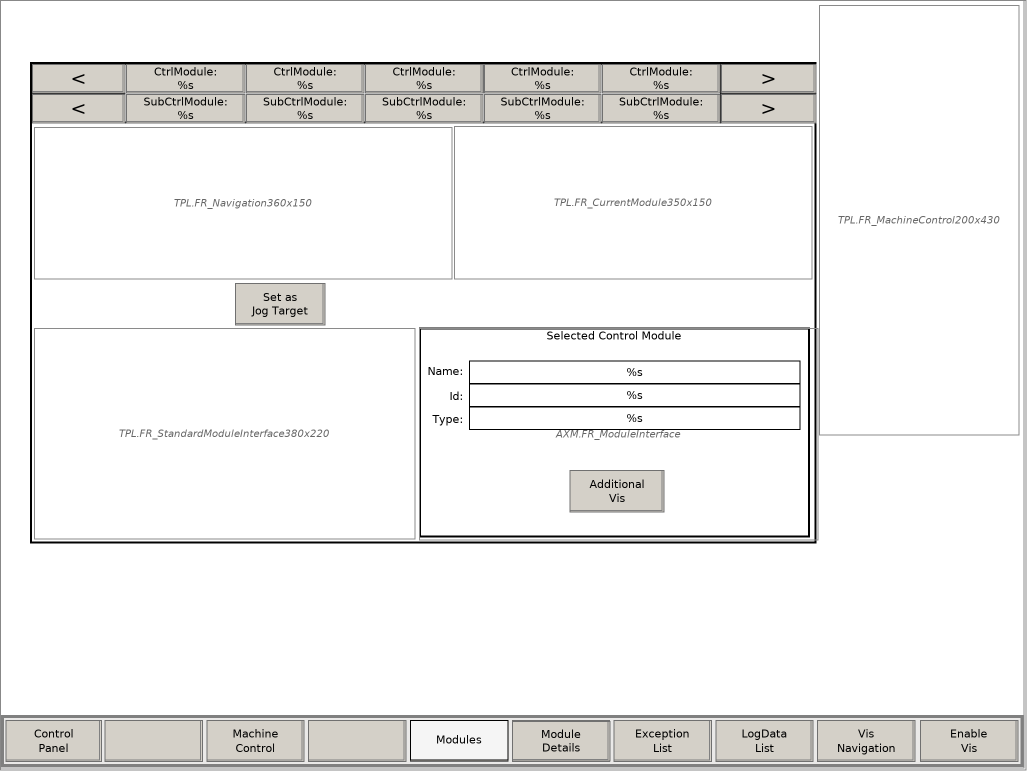
VISUALIZATION VIS_Modules  // 1027x771
    Frame (0,0 1024x768)
        shows TPL.FR_Nav1024x768(i_sTitle := 'Template: Modules')
    Frame (1,715 1024x54)
        shows FR_NavigationButtons()
    Rectangle (30,62 786x481)
    Rectangle (30,63 786x60)
    Button (602,64 118x29), "EQModule: %s", tooltip "%s", text variable: SR_VisControl.vpq_audiIdModuleList[5], colour toggle: SR_VisControl.vpq_axActiveModuleList[5], invisible if: SR_VisControl.vpq_axDisableModuleList[5] OR SR_VisControl.vpq_axIdModuleListValid[5] = FALSE, input disabled if: SR_VisControl.vpq_axDisableModuleList[5]
        p4168582468: SR_VisControl.vpq_asNameModuleList[5]
        toggle SR_VisControl.vpiq_axModuleList[5]
    Button (483,64 118x29), "EQModule: %s", tooltip "%s", text variable: SR_VisControl.vpq_audiIdModuleList[4], colour toggle: SR_VisControl.vpq_axActiveModuleList[4], invisible if: SR_VisControl.vpq_axDisableModuleList[4] OR SR_VisControl.vpq_axIdModuleListValid[4] = FALSE, input disabled if: SR_VisControl.vpq_axDisableModuleList[4]
        p4168582468: SR_VisControl.vpq_asNameModuleList[4]
        toggle SR_VisControl.vpiq_axModuleList[4]
    Button (365,64 118x29), "EQModule: %s", tooltip "%s", text variable: SR_VisControl.vpq_audiIdModuleList[3], colour toggle: SR_VisControl.vpq_axActiveModuleList[3], invisible if: SR_VisControl.vpq_axDisableModuleList[3] OR SR_VisControl.vpq_axIdModuleListValid[3] = FALSE, input disabled if: SR_VisControl.vpq_axDisableModuleList[3]
        p4168582468: SR_VisControl.vpq_asNameModuleList[3]
        toggle SR_VisControl.vpiq_axModuleList[3]
    Button (246,64 118x29), "EQModule: %s", tooltip "%s", text variable: SR_VisControl.vpq_audiIdModuleList[2], colour toggle: SR_VisControl.vpq_axActiveModuleList[2], invisible if: SR_VisControl.vpq_axDisableModuleList[2] OR SR_VisControl.vpq_axIdModuleListValid[2] = FALSE, input disabled if: SR_VisControl.vpq_axDisableModuleList[2]
        p4168582468: SR_VisControl.vpq_asNameModuleList[2]
        toggle SR_VisControl.vpiq_axModuleList[2]
    Button (126,64 119x29), "EQModule: %s", tooltip "%s", text variable: SR_VisControl.vpq_audiIdModuleList[1], colour toggle: SR_VisControl.vpq_axActiveModuleList[1], invisible if: SR_VisControl.vpq_axDisableModuleList[1] OR SR_VisControl.vpq_axIdModuleListValid[1] = FALSE, input disabled if: SR_VisControl.vpq_axDisableModuleList[1]
        p4168582468: SR_VisControl.vpq_asNameModuleList[1]
        toggle SR_VisControl.vpiq_axModuleList[1]
    Button (126,94 119x29), "SubEQModule: %s", tooltip "%s", text variable: SR_VisControl.vpq_audiIdSubModuleList[1], colour toggle: SR_VisControl.vpq_axActiveSubModuleList[1], invisible if: SR_VisControl.vpq_axDisableSubModuleList[1] OR SR_VisControl.vpq_axIdSubModuleListValid[1] = FALSE, input disabled if: SR_VisControl.vpq_axDisableSubModuleList[1]
        p4168582468: SR_VisControl.vpq_asNameSubModuleList[1]
        toggle SR_VisControl.vpiq_axSubModuleList[1]
    Button (246,94 118x29), "SubEQModule: %s", tooltip "%s", text variable: SR_VisControl.vpq_audiIdSubModuleList[2], colour toggle: SR_VisControl.vpq_axActiveSubModuleList[2], invisible if: SR_VisControl.vpq_axDisableSubModuleList[2] OR SR_VisControl.vpq_axIdSubModuleListValid[2] = FALSE, input disabled if: SR_VisControl.vpq_axDisableSubModuleList[2]
        p4168582468: SR_VisControl.vpq_asNameSubModuleList[2]
        toggle SR_VisControl.vpiq_axSubModuleList[2]
    Button (365,94 118x29), "SubEQModule: %s", tooltip "%s", text variable: SR_VisControl.vpq_audiIdSubModuleList[3], colour toggle: SR_VisControl.vpq_axActiveSubModuleList[3], invisible if: SR_VisControl.vpq_axDisableSubModuleList[3] OR SR_VisControl.vpq_axIdSubModuleListValid[3] = FALSE, input disabled if: SR_VisControl.vpq_axDisableSubModuleList[3]
        p4168582468: SR_VisControl.vpq_asNameSubModuleList[3]
        toggle SR_VisControl.vpiq_axSubModuleList[3]
    Button (484,94 117x29), "SubEQModule: %s", tooltip "%s", text variable: SR_VisControl.vpq_audiIdSubModuleList[4], colour toggle: SR_VisControl.vpq_axActiveSubModuleList[4], invisible if: SR_VisControl.vpq_axDisableSubModuleList[4] OR SR_VisControl.vpq_axIdSubModuleListValid[4] = FALSE, input disabled if: SR_VisControl.vpq_axDisableSubModuleList[4]
        p4168582468: SR_VisControl.vpq_asNameSubModuleList[4]
        toggle SR_VisControl.vpiq_axSubModuleList[4]
    Button (602,94 118x29), "SubEQModule: %s", tooltip "%s", text variable: SR_VisControl.vpq_audiIdSubModuleList[5], colour toggle: SR_VisControl.vpq_axActiveSubModuleList[5], invisible if: SR_VisControl.vpq_axDisableSubModuleList[5] OR SR_VisControl.vpq_axIdSubModuleListValid[5] = FALSE, input disabled if: SR_VisControl.vpq_axDisableSubModuleList[5]
        p4168582468: SR_VisControl.vpq_asNameSubModuleList[5]
        toggle SR_VisControl.vpiq_axSubModuleList[5]
    Rectangle (720,93 95x29), ">"
    Rectangle (720,63 95x30), ">"
    Button (721,64 95x29), ">", invisible if: SR_VisControl.vpq_xDisableModuleListUp, input disabled if: SR_VisControl.vpq_xDisableModuleListUp
        toggle SR_VisControl.vpiq_xModuleListUp
    Button (721,94 95x29), ">", invisible if: SR_VisControl.vpq_xDisableSubModuleListUp, input disabled if: SR_VisControl.vpq_xDisableSubModuleListUp
        toggle SR_VisControl.vpiq_xSubModuleListUp
    Rectangle (31,93 94x29), "<"
    Rectangle (31,64 94x30), "<"
    Button (32,64 93x29), "<", invisible if: SR_VisControl.vpq_xDisableModuleListDown, input disabled if: SR_VisControl.vpq_xDisableModuleListDown
        toggle SR_VisControl.vpiq_xModuleListDown
    Button (32,94 93x29), "<", invisible if: SR_VisControl.vpq_xDisableSubModuleListDown, input disabled if: SR_VisControl.vpq_xDisableSubModuleListDown
        toggle SR_VisControl.vpiq_xSubModuleListDown
    Button (235,283 90x42), "Set as Jog Target", colour toggle: SR_VisControl.vpq_xCurrentIsJogTarget, invisible if: SR_VisControl.vpq_xButtonSetJogTargetInvisible
        tap SR_VisControl.vpiq_xButtonSetCurrentAsJogTarget
    Frame (34,127 418x152)
        shows TPL.FR_Navigation360x150(i_sNameNavRight := SR_VisControl.vpq_sNameNavRight, i_sNameNavUp := SR_VisControl.vpq_sNameNavUp, i_sNameNavLeft := SR_VisControl.vpq_sNameNavLeft, i_sNameNavDown := SR_VisControl.vpq_sNameNavDown, i_xEnableNavUp := SR_VisControl.vpq_xEnableNavUp, i_xEnableNavLeft := SR_VisControl.vpq_xEnableNavLeft, i_xEnableNavRight := SR_VisControl.vpq_xEnableNavRight, i_xEnableNavDown := SR_VisControl.vpq_xEnableNavDown, iq_xNavUp := SR_VisControl.vpiq_xNavUp, iq_xNavLeft := SR_VisControl.vpiq_xNavLeft, iq_xNavRight := SR_VisControl.vpiq_xNavRight, iq_xNavDown := SR_VisControl.vpiq_xNavDown)
    Frame (454,126 358x153)
        shows TPL.FR_CurrentModule350x150(i_stCurrentModuleStandardItf := SR_VisControl.vpq_stCurrentModuleStandardInterface)
        p2332068554: SR_VisControl.stCurrentModuleStandardInterface
        p427866952: SR_VisControl.stCurrentModuleStandardInterface
        p2190627833: SR_VisControl.vpq_stCurrentModuleStandardInterface
    Button (126,64 119x29), "CtrlModule: %s", tooltip "%s", text variable: SR_VisControl.vpq_asControlModuleButtonName[1], colour toggle: SR_VisControl.vpq_axControlModuleActive[1], invisible if: SR_VisControl.vpq_axControlModuleValid[1]=FALSE
        p4168582468: SR_VisControl.vpq_asToolTipControlModuleList[1]
        toggle SR_VisControl.vpiq_axControlModuleList[1]
    Button (246,64 118x29), "CtrlModule: %s", tooltip "%s", text variable: SR_VisControl.vpq_asControlModuleButtonName[2], colour toggle: SR_VisControl.vpq_axControlModuleActive[2], invisible if: SR_VisControl.vpq_axControlModuleValid[2]=FALSE
        p4168582468: SR_VisControl.vpq_asToolTipControlModuleList[2]
        toggle SR_VisControl.vpiq_axControlModuleList[2]
    Button (365,64 118x29), "CtrlModule: %s", tooltip "%s", text variable: SR_VisControl.vpq_asControlModuleButtonName[3], colour toggle: SR_VisControl.vpq_axControlModuleActive[3], invisible if: SR_VisControl.vpq_axControlModuleValid[3]=FALSE
        p4168582468: SR_VisControl.vpq_asToolTipControlModuleList[3]
        toggle SR_VisControl.vpiq_axControlModuleList[3]
    Button (484,64 117x29), "CtrlModule: %s", tooltip "%s", text variable: SR_VisControl.vpq_asControlModuleButtonName[4], colour toggle: SR_VisControl.vpq_axControlModuleActive[4], invisible if: SR_VisControl.vpq_axControlModuleValid[4]=FALSE
        p4168582468: SR_VisControl.vpq_asToolTipControlModuleList[4]
        toggle SR_VisControl.vpiq_axControlModuleList[4]
    Button (602,64 118x29), "CtrlModule: %s", tooltip "%s", text variable: SR_VisControl.vpq_asControlModuleButtonName[5], colour toggle: SR_VisControl.vpq_axControlModuleActive[5], invisible if: SR_VisControl.vpq_axControlModuleValid[5]=FALSE
        p4168582468: SR_VisControl.vpq_asToolTipControlModuleList[5]
        toggle SR_VisControl.vpiq_axControlModuleList[5]
    Button (126,94 119x29), "SubCtrlModule: %s", tooltip "%s", text variable: SR_VisControl.vpq_asSubControlModuleButtonName[1], colour toggle: SR_VisControl.vpq_axSubControlModuleActive[1], invisible if: SR_VisControl.vpq_axSubControlModuleValid[1]=FALSE
        p4168582468: SR_VisControl.vpq_asToolTipSubControlModuleList[1]
        toggle SR_VisControl.vpiq_axSubControlModuleList[1]
    Button (246,94 118x29), "SubCtrlModule: %s", tooltip "%s", text variable: SR_VisControl.vpq_asSubControlModuleButtonName[2], colour toggle: SR_VisControl.vpq_axSubControlModuleActive[2], invisible if: SR_VisControl.vpq_axSubControlModuleValid[2]=FALSE
        p4168582468: SR_VisControl.vpq_asToolTipSubControlModuleList[2]
        toggle SR_VisControl.vpiq_axSubControlModuleList[2]
    Button (365,94 118x29), "SubCtrlModule: %s", tooltip "%s", text variable: SR_VisControl.vpq_asSubControlModuleButtonName[3], colour toggle: SR_VisControl.vpq_axSubControlModuleActive[3], invisible if: SR_VisControl.vpq_axSubControlModuleValid[3]=FALSE
        p4168582468: SR_VisControl.vpq_asToolTipSubControlModuleList[3]
        toggle SR_VisControl.vpiq_axSubControlModuleList[3]
    Button (484,94 117x29), "SubCtrlModule: %s", tooltip "%s", text variable: SR_VisControl.vpq_asSubControlModuleButtonName[4], colour toggle: SR_VisControl.vpq_axSubControlModuleActive[4], invisible if: SR_VisControl.vpq_axSubControlModuleValid[4]=FALSE
        p4168582468: SR_VisControl.vpq_asToolTipSubControlModuleList[4]
        toggle SR_VisControl.vpiq_axSubControlModuleList[4]
    Button (602,94 118x29), "SubCtrlModule: %s", tooltip "%s", text variable: SR_VisControl.vpq_asSubControlModuleButtonName[5], colour toggle: SR_VisControl.vpq_axSubControlModuleActive[5], invisible if: SR_VisControl.vpq_axSubControlModuleValid[5]=FALSE
        p4168582468: SR_VisControl.vpq_asToolTipSubControlModuleList[5]
        toggle SR_VisControl.vpiq_axSubControlModuleList[5]
    Frame (418,327 394x212), invisible if: SR_VisControl.vpq_udiActiveControlModuleNumber <> 0
        shows FR_OtherModuleTypes()
    Frame (418,327 394x212), invisible if: SR_VisControl.vpq_udiActiveControlModuleNumber = 0
        shows FR_ControlModuleTypes(i_sControlModuleName := SR_VisControl.stCurrentControlModuleStandardInterface.sControlModuleName, i_diControlModuleNumber := TO_DINT(SR_VisControl.stCurrentControlModuleStandardInterface.udiControlModuleNumber), i_diControlModuleType := TO_DINT(SR_VisControl.stCurrentControlModuleStandardInterface.udiControlModuleType))
        p159172089: SR_VisControl.IFB_AxisModuleVisController
        p2210332906: SR_VisControl.IFB_AxisModuleVisController.iPaneSelect
    Frame (34,328 381x211)
        shows TPL.FR_StandardModuleInterface380x220(i_stCurrentModuleStandardItf := SR_VisControl.vpq_stCurrentModuleStandardInterface, i_sCurrentModuleReaction := SR_VisControl.vpq_sCurrentModuleReaction, i_udiModuleReactionIndexMin := SR_VisControl.vpq_udiModuleReactionIndexMin, i_axModuleReaction := SR_VisControl.vpq_axModuleReaction, i_udiNumberOfReactions := TPL.Gc_udiMaxNumberOfReactions, iq_xModuleReactionDown := SR_VisControl.vpiq_xModuleReactionDown, iq_xModuleReactionUp := SR_VisControl.vpiq_xModuleReactionUp, iq_diStartStepToSet := SR_VisControl.vpiq_diStartStepToSet, iq_diCmdToSet := SR_VisControl.vpiq_diCmdToSet, iq_xEnableModuleClicked := SR_VisControl.vpiq_xEnableModuleClicked, iq_xSetCmdClicked := SR_VisControl.vpiq_xSetCmdClicked, iq_fbVisContExHandling := SR_VisControl.vpiq_fbVisContExHandling)
        p1094400588: SR_VisControl.IFB_AxisModuleVisController.xCurrentIsOfMyType
        p3339340907: 'Vis_ModuleError'
        p1029787830: SR_VisControl.vpiq_fbVisContExHandling
        p2258115317: SR_VisControl.iModuleErrorReactionIndexMin
        p2777435286: SR_VisControl.axModuleErrorReaction
        p214250784: TPC_Gc_diMaxNumberOfErrorReactions
        p311732222: SR_VisControl.stCurrentModuleStandardInterface
        p640132070: SR_VisControl.xModuleErrorReactionDown
        p4234372197: SR_VisControl.xModuleErrorReactionUp
        p2938682392: SR_VisControl.xEnableModule_Clicked
        p3592490199: SR_VisControl.xSetCmd_Clicked
        p2560461379: SR_VisControl.diStartStepToSet
        p2307280719: SR_VisControl.stCurrentModuleStandardInterface
        p2190627833: SR_VisControl.vpq_stCurrentModuleStandardInterface
    Frame (419,328 399x212), invisible if: SR_VisControl.vpq_stCurrentModuleStandardInterface.q_dwModuleType <> 3
        shows AXM.FR_ModuleInterface(iq_fbAxisModuleVisController := SR_VisControl.vpiq_fbAxisModuleVisController)
        p159172089: SR_VisControl.IFB_AxisModuleVisController
        p2210332906: SR_VisControl.IFB_AxisModuleVisController.iPaneSelect
        p856915466: SR_VisControl.stCurrentControlModuleStandardInterface.udiControlModuleNumber
        p2344652976: SR_VisControl.stCurrentControlModuleStandardInterface.udiControlModuleType
        p467735965: SR_VisControl.stCurrentControlModuleStandardInterface.sControlModuleName
    Button (512,721 98x40), "Module Details"
        OnMouseClick:  Assign=VIS_ModuleDetails, Type=Assignment
    Rectangle (410,720 98x40), "Modules"
    Frame (819,5 200x430), invisible if: NOT SR_VisControl.vpiq_xShowControlFrame
        shows TPL.FR_MachineControl200x430(i_stMachineItf := SR_VisControl.vpq_stMachineInterface, i_xPrepareActive := G_xPrepareActive, i_xAutoActive := G_xAutoActive, i_xBrakeReleaseActive := G_xBrakeReleaseActive, i_xJogMachineActive := G_xJogMachineActive, i_xManualActive := G_xManualActive, i_xException := SR_VisControl.vpq_xMachineInException, i_dwDiagQuitColor := SR_VisControl.vpq_dwDiagQuitColor, iq_iPositionX := SR_VisControl.vpiq_iPositionX, iq_iPositionY := SR_VisControl.vpiq_iPositionY, iq_xEmergencyEpas := G_xEmergencyEpas, iq_xStartEpas := G_xStartEpas, iq_xStopEpas := G_xStopEpas, iq_xJogForwEpas := G_xJogForwEpas, iq_xJogBackEpas := G_xJogBackEpas, iq_xDoPrepare := G_xDoPrepare, iq_xDoAuto := G_xDoAuto, iq_xDoBrakeRelease := G_xDoBrakeRelease, iq_xDoJogMachine := G_xDoJogMachine, iq_xDoManual := G_xDoManual, iq_xDiagQuitEpas := G_xDiagQuitEpas)
        p1457045297: SR_VisControl.stMachineInterface.stQ.xError
        p1941967854: g_I_xEmergency_Epas
        p2531571229: g_I_xStart_Epas
        p1511842254: g_I_xStop_Epas
        p745511063: g_I_xJogForw_Epas
        p3518271027: g_I_xJogBack_Epas
        p1982879521: g_I_xErrorQuit_Epas
        p3866886353: SR_VisControl.dwErrorQuitColor
        p1761348311: SR_VisControl.vpq_stMachineInterface
        p3560616238: SR_VisControl.vpiq_iPositionX
        p2738717112: SR_VisControl.vpiq_iPositionY
END_VISUALIZATION

